gfCNCPoint4[13273] = {X 270.8909, Y 44.1700, Z -5.5000, A 0.000, B 0.000, C 0.000 }
gfCNCPoint4[13274] = {X 270.8910, Y 45.0000, Z -5.5000, A 0.000, B 0.000, C 0.000 }
gfCNCPoint4[13275] = {X 270.7867, Y 45.9257, Z -5.5000, A 0.000, B 0.000, C 0.000 }
gfCNCPoint4[13276] = {X 270.4791, Y 46.8050, Z -5.5000, A 0.000, B 0.000, C 0.000 }
gfCNCPoint4[13277] = {X 269.9835, Y 47.5937, Z -5.5000, A 0.000, B 0.000, C 0.000 }
gfCNCPoint4[13278] = {X 269.3247, Y 48.2524, Z -5.5000, A 0.000, B 0.000, C 0.000 }
gfCNCPoint4[13279] = {X 268.5360, Y 48.7480, Z -5.5000, A 0.000, B 0.000, C 0.000 }
gfCNCPoint4[13280] = {X 267.6567, Y 49.0557, Z -5.5000, A 0.000, B 0.000, C 0.000 }
gfCNCPoint4[13281] = {X 266.7310, Y 49.1600, Z -5.5000, A 0.000, B 0.000, C 0.000 }
gfCNCPoint4[13282] = {X 260.2876, Y 49.1600, Z -5.5000, A 0.000, B 0.000, C 0.000 }
gfCNCPoint4[13283] = {X 259.3664, Y 49.0567, Z -5.5000, A 0.000, B 0.000, C 0.000 }
gfCNCPoint4[13284] = {X 258.4910, Y 48.7520, Z -5.5000, A 0.000, B 0.000, C 0.000 }
gfCNCPoint4[13285] = {X 257.7047, Y 48.2611, Z -5.5000, A 0.000, B 0.000, C 0.000 }
gfCNCPoint4[13286] = {X 257.0467, Y 47.6082, Z -5.5000, A 0.000, B 0.000, C 0.000 }
gfCNCPoint4[13287] = {X 256.5496, Y 46.8258, Z -5.5000, A 0.000, B 0.000, C 0.000 }
gfCNCPoint4[13288] = {X 256.2381, Y 45.9527, Z -5.5000, A 0.000, B 0.000, C 0.000 }
gfCNCPoint4[13289] = {X 256.1277, Y 45.0324, Z -5.5000, A 0.000, B 0.000, C 0.000 }
gfCNCPoint4[13290] = {X 256.1280, Y 44.1516, Z -5.5000, A 0.000, B 0.000, C 0.000 }
gfCNCPoint4[13291] = {X 256.2385, Y 43.2545, Z -5.5000, A 0.000, B 0.000, C 0.000 }
gfCNCPoint4[13292] = {X 256.5401, Y 42.4026, Z -5.5000, A 0.000, B 0.000, C 0.000 }
gfCNCPoint4[13293] = {X 257.0187, Y 41.6358, Z -5.5000, A 0.000, B 0.000, C 0.000 }
gfCNCPoint4[13294] = {X 257.6515, Y 40.9906, Z -5.5000, A 0.000, B 0.000, C 0.000 }
gfCNCPoint4[13295] = {X 257.6515, Y 34.3138, Z -5.5000, A 0.000, B 0.000, C 0.000 }
gfCNCPoint4[13296] = {X 254.6703, Y 34.3138, Z -5.5000, A 0.000, B 0.000, C 0.000 }
gfCNCPoint4[13297] = {X 250.3102, Y 42.8068, Z -5.5000, A 0.000, B 0.000, C 0.000 }
gfCNCPoint4[13298] = {X 250.4892, Y 43.4800, Z -5.5000, A 0.000, B 0.000, C 0.000 }
gfCNCPoint4[13299] = {X 250.5534, Y 44.1736, Z -5.5000, A 0.000, B 0.000, C 0.000 }
gfCNCPoint4[13300] = {X 250.5536, Y 45.0000, Z -5.5000, A 0.000, B 0.000, C 0.000 }
gfCNCPoint4[13301] = {X 250.4493, Y 45.9257, Z -5.5000, A 0.000, B 0.000, C 0.000 }
gfCNCPoint4[13302] = {X 250.1416, Y 46.8050, Z -5.5000, A 0.000, B 0.000, C 0.000 }
gfCNCPoint4[13303] = {X 249.6460, Y 47.5937, Z -5.5000, A 0.000, B 0.000, C 0.000 }
gfCNCPoint4[13304] = {X 248.9873, Y 48.2524, Z -5.5000, A 0.000, B 0.000, C 0.000 }
gfCNCPoint4[13305] = {X 248.1985, Y 48.7480, Z -5.5000, A 0.000, B 0.000, C 0.000 }
gfCNCPoint4[13306] = {X 247.3192, Y 49.0557, Z -5.5000, A 0.000, B 0.000, C 0.000 }
gfCNCPoint4[13307] = {X 246.3936, Y 49.1600, Z -5.5000, A 0.000, B 0.000, C 0.000 }
gfCNCPoint4[13308] = {X 239.8075, Y 49.1600, Z -5.5000, A 0.000, B 0.000, C 0.000 }
gfCNCPoint4[13309] = {X 238.8818, Y 49.0557, Z -5.5000, A 0.000, B 0.000, C 0.000 }
gfCNCPoint4[13310] = {X 238.0026, Y 48.7480, Z -5.5000, A 0.000, B 0.000, C 0.000 }
gfCNCPoint4[13311] = {X 237.2138, Y 48.2524, Z -5.5000, A 0.000, B 0.000, C 0.000 }
gfCNCPoint4[13312] = {X 236.5551, Y 47.5937, Z -5.5000, A 0.000, B 0.000, C 0.000 }
gfCNCPoint4[13313] = {X 236.0595, Y 46.8050, Z -5.5000, A 0.000, B 0.000, C 0.000 }
gfCNCPoint4[13314] = {X 235.7518, Y 45.9257, Z -5.5000, A 0.000, B 0.000, C 0.000 }
gfCNCPoint4[13315] = {X 235.6475, Y 45.0000, Z -5.5000, A 0.000, B 0.000, C 0.000 }
gfCNCPoint4[13316] = {X 235.6479, Y 44.1516, Z -5.5000, A 0.000, B 0.000, C 0.000 }
gfCNCPoint4[13317] = {X 235.7441, Y 43.3174, Z -5.5000, A 0.000, B 0.000, C 0.000 }
gfCNCPoint4[13318] = {X 236.0059, Y 42.5195, Z -5.5000, A 0.000, B 0.000, C 0.000 }
gfCNCPoint4[13319] = {X 236.4226, Y 41.7905, Z -5.5000, A 0.000, B 0.000, C 0.000 }
gfCNCPoint4[13320] = {X 236.9772, Y 41.1600, Z -5.5000, A 0.000, B 0.000, C 0.000 }
gfCNCPoint4[13321] = {X 237.6471, Y 40.6537, Z -5.5000, A 0.000, B 0.000, C 0.000 }
gfCNCPoint4[13322] = {X 238.4051, Y 40.2923, Z -5.5000, A 0.000, B 0.000, C 0.000 }
gfCNCPoint4[13323] = {X 242.4918, Y 32.2930, Z -5.5000, A 0.000, B 0.000, C 0.000 }
gfCNCPoint4[13324] = {X 241.3078, Y 31.5182, Z -5.5000, A 0.000, B 0.000, C 0.000 }
gfCNCPoint4[13325] = {X 240.2313, Y 30.5999, Z -5.5000, A 0.000, B 0.000, C 0.000 }
gfCNCPoint4[13326] = {X 239.2796, Y 29.5527, Z -5.5000, A 0.000, B 0.000, C 0.000 }
gfCNCPoint4[13327] = {X 238.4681, Y 28.3935, Z -5.5000, A 0.000, B 0.000, C 0.000 }
gfCNCPoint4[13328] = {X 237.8099, Y 27.1410, Z -5.5000, A 0.000, B 0.000, C 0.000 }
gfCNCPoint4[13329] = {X 237.3154, Y 25.8152, Z -5.5000, A 0.000, B 0.000, C 0.000 }
gfCNCPoint4[13330] = {X 236.8995, Y 24.0215, Z -5.5000, A 0.000, B 0.000, C 0.000 }
gfCNCPoint4[13331] = {X 236.6876, Y 22.1924, Z -5.5000, A 0.000, B 0.000, C 0.000 }
gfCNCPoint4[13332] = {X 236.6824, Y 20.3512, Z -5.5000, A 0.000, B 0.000, C 0.000 }
gfCNCPoint4[13333] = {X 236.8839, Y 18.5210, Z -5.5000, A 0.000, B 0.000, C 0.000 }
gfCNCPoint4[13334] = {X 237.2897, Y 16.7249, Z -5.5000, A 0.000, B 0.000, C 0.000 }
gfCNCPoint4[13335] = {X 237.8524, Y 15.1703, Z -5.5000, A 0.000, B 0.000, C 0.000 }
gfCNCPoint4[13336] = {X 238.6289, Y 13.7107, Z -5.5000, A 0.000, B 0.000, C 0.000 }
gfCNCPoint4[13337] = {X 239.6035, Y 12.3752, Z -5.5000, A 0.000, B 0.000, C 0.000 }
gfCNCPoint4[13338] = {X 240.7569, Y 11.1905, Z -5.5000, A 0.000, B 0.000, C 0.000 }
gfCNCPoint4[13339] = {X 242.0658, Y 10.1805, Z -5.5000, A 0.000, B 0.000, C 0.000 }
gfCNCPoint4[13340] = {X 243.5041, Y 9.3652, Z -5.5000, A 0.000, B 0.000, C 0.000 }
gfCNCPoint4[13341] = {X 245.0431, Y 8.7610, Z -5.5000, A 0.000, B 0.000, C 0.000 }
gfCNCPoint4[13342] = {X 246.6520, Y 8.3800, Z -5.5000, A 0.000, B 0.000, C 0.000 }
gfCNCPoint4[13343] = {X 248.7352, Y 8.1102, Z -5.5000, A 0.000, B 0.000, C 0.000 }
gfCNCPoint4[13344] = {X 250.8343, Y 8.0302, Z -5.5000, A 0.000, B 0.000, C 0.000 }
gfCNCPoint4[13345] = {X 266.7621, Y 8.0302, Z -5.5000, A 0.000, B 0.000, C 0.000 }
gfCNCPoint4[13346] = {X 267.6819, Y 8.1408, Z -5.5000, A 0.000, B 0.000, C 0.000 }
gfCNCPoint4[13347] = {X 268.5546, Y 8.4520, Z -5.5000, A 0.000, B 0.000, C 0.000 }
gfCNCPoint4[13348] = {X 269.3368, Y 8.9486, Z -5.5000, A 0.000, B 0.000, C 0.000 }
gfCNCPoint4[13349] = {X 269.9897, Y 9.6059, Z -5.5000, A 0.000, B 0.000, C 0.000 }
gfCNCPoint4[13350] = {X 270.4811, Y 10.3913, Z -5.5000, A 0.000, B 0.000, C 0.000 }
gfCNCPoint4[13351] = {X 270.7866, Y 11.2660, Z -5.5000, A 0.000, B 0.000, C 0.000 }
gfCNCPoint4[13352] = {X 270.8910, Y 12.1866, Z -5.5000, A 0.000, B 0.000, C 0.000 }
gfCNCPoint4[13353] = {X 270.8908, Y 13.0208, Z -5.5000, A 0.000, B 0.000, C 0.000 }
gfCNCPoint4[13354] = {X 270.7824, Y 13.9226, Z -5.5000, A 0.000, B 0.000, C 0.000 }
gfCNCPoint4[13355] = {X 270.4808, Y 14.7793, Z -5.5000, A 0.000, B 0.000, C 0.000 }
gfCNCPoint4[13356] = {X 270.0005, Y 15.5502, Z -5.5000, A 0.000, B 0.000, C 0.000 }
gfCNCPoint4[13357] = {X 269.3643, Y 16.1985, Z -5.5000, A 0.000, B 0.000, C 0.000 }
gfCNCPoint4[13358] = {X 269.3642, Y 28.5936, Z -5.5000, A 0.000, B 0.000, C 0.000 }
gfCNCPoint4[13359] = {X 273.3642, Y 28.5936, Z -5.5000, A 0.000, B 0.000, C 0.000 }
gfCNCPoint4[13360] = {X 269.2842, Y 28.5936, Z -5.5000, A 0.000, B 0.000, C 0.000 }
gfCNCPoint4[13361] = {X 269.2842, Y 41.0277, Z -5.5000, A 0.000, B 0.000, C 0.000 }
gfCNCPoint4[13362] = {X 269.3838, Y 41.1089, Z -5.5000, A 0.000, B 0.000, C 0.000 }
gfCNCPoint4[13363] = {X 269.9802, Y 41.7411, Z -5.5000, A 0.000, B 0.000, C 0.000 }
gfCNCPoint4[13364] = {X 270.4291, Y 42.4852, Z -5.5000, A 0.000, B 0.000, C 0.000 }
gfCNCPoint4[13365] = {X 270.7103, Y 43.3076, Z -5.5000, A 0.000, B 0.000, C 0.000 }
gfCNCPoint4[13366] = {X 270.8109, Y 44.1708, Z -5.5000, A 0.000, B 0.000, C 0.000 }
gfCNCPoint4[13367] = {X 270.8110, Y 45.0000, Z -5.5000, A 0.000, B 0.000, C 0.000 }
gfCNCPoint4[13368] = {X 270.7087, Y 45.9079, Z -5.5000, A 0.000, B 0.000, C 0.000 }
gfCNCPoint4[13369] = {X 270.4070, Y 46.7702, Z -5.5000, A 0.000, B 0.000, C 0.000 }
gfCNCPoint4[13370] = {X 269.9209, Y 47.5438, Z -5.5000, A 0.000, B 0.000, C 0.000 }
gfCNCPoint4[13371] = {X 269.2749, Y 48.1899, Z -5.5000, A 0.000, B 0.000, C 0.000 }
gfCNCPoint4[13372] = {X 268.5013, Y 48.6760, Z -5.5000, A 0.000, B 0.000, C 0.000 }
gfCNCPoint4[13373] = {X 267.6389, Y 48.9777, Z -5.5000, A 0.000, B 0.000, C 0.000 }
gfCNCPoint4[13374] = {X 266.7310, Y 49.0800, Z -5.5000, A 0.000, B 0.000, C 0.000 }
gfCNCPoint4[13375] = {X 260.2876, Y 49.0800, Z -5.5000, A 0.000, B 0.000, C 0.000 }
gfCNCPoint4[13376] = {X 259.3841, Y 48.9787, Z -5.5000, A 0.000, B 0.000, C 0.000 }
gfCNCPoint4[13377] = {X 258.5255, Y 48.6799, Z -5.5000, A 0.000, B 0.000, C 0.000 }
gfCNCPoint4[13378] = {X 257.7544, Y 48.1983, Z -5.5000, A 0.000, B 0.000, C 0.000 }
gfCNCPoint4[13379] = {X 257.1090, Y 47.5580, Z -5.5000, A 0.000, B 0.000, C 0.000 }
gfCNCPoint4[13380] = {X 256.6215, Y 46.7907, Z -5.5000, A 0.000, B 0.000, C 0.000 }
gfCNCPoint4[13381] = {X 256.3160, Y 45.9344, Z -5.5000, A 0.000, B 0.000, C 0.000 }
gfCNCPoint4[13382] = {X 256.2077, Y 45.0318, Z -5.5000, A 0.000, B 0.000, C 0.000 }
gfCNCPoint4[13383] = {X 256.2080, Y 44.1527, Z -5.5000, A 0.000, B 0.000, C 0.000 }
gfCNCPoint4[13384] = {X 256.3185, Y 43.2637, Z -5.5000, A 0.000, B 0.000, C 0.000 }
gfCNCPoint4[13385] = {X 256.6204, Y 42.4203, Z -5.5000, A 0.000, B 0.000, C 0.000 }
gfCNCPoint4[13386] = {X 257.0991, Y 41.6631, Z -5.5000, A 0.000, B 0.000, C 0.000 }
gfCNCPoint4[13387] = {X 257.7315, Y 41.0287, Z -5.5000, A 0.000, B 0.000, C 0.000 }
gfCNCPoint4[13388] = {X 257.7315, Y 34.2338, Z -5.5000, A 0.000, B 0.000, C 0.000 }
gfCNCPoint4[13389] = {X 254.6215, Y 34.2338, Z -5.5000, A 0.000, B 0.000, C 0.000 }
gfCNCPoint4[13390] = {X 250.2231, Y 42.8013, Z -5.5000, A 0.000, B 0.000, C 0.000 }
gfCNCPoint4[13391] = {X 250.4074, Y 43.4770, Z -5.5000, A 0.000, B 0.000, C 0.000 }
gfCNCPoint4[13392] = {X 250.4734, Y 44.1743, Z -5.5000, A 0.000, B 0.000, C 0.000 }
gfCNCPoint4[13393] = {X 250.4736, Y 45.0000, Z -5.5000, A 0.000, B 0.000, C 0.000 }
gfCNCPoint4[13394] = {X 250.3713, Y 45.9079, Z -5.5000, A 0.000, B 0.000, C 0.000 }
gfCNCPoint4[13395] = {X 250.0695, Y 46.7702, Z -5.5000, A 0.000, B 0.000, C 0.000 }
gfCNCPoint4[13396] = {X 249.5834, Y 47.5438, Z -5.5000, A 0.000, B 0.000, C 0.000 }
gfCNCPoint4[13397] = {X 248.9374, Y 48.1899, Z -5.5000, A 0.000, B 0.000, C 0.000 }
gfCNCPoint4[13398] = {X 248.1638, Y 48.6760, Z -5.5000, A 0.000, B 0.000, C 0.000 }
gfCNCPoint4[13399] = {X 247.3014, Y 48.9777, Z -5.5000, A 0.000, B 0.000, C 0.000 }
gfCNCPoint4[13400] = {X 246.3936, Y 49.0800, Z -5.5000, A 0.000, B 0.000, C 0.000 }
gfCNCPoint4[13401] = {X 239.8075, Y 49.0800, Z -5.5000, A 0.000, B 0.000, C 0.000 }
gfCNCPoint4[13402] = {X 238.8996, Y 48.9777, Z -5.5000, A 0.000, B 0.000, C 0.000 }
gfCNCPoint4[13403] = {X 238.0373, Y 48.6760, Z -5.5000, A 0.000, B 0.000, C 0.000 }
gfCNCPoint4[13404] = {X 237.2637, Y 48.1899, Z -5.5000, A 0.000, B 0.000, C 0.000 }
gfCNCPoint4[13405] = {X 236.6176, Y 47.5438, Z -5.5000, A 0.000, B 0.000, C 0.000 }
gfCNCPoint4[13406] = {X 236.1315, Y 46.7702, Z -5.5000, A 0.000, B 0.000, C 0.000 }
gfCNCPoint4[13407] = {X 235.8298, Y 45.9079, Z -5.5000, A 0.000, B 0.000, C 0.000 }
gfCNCPoint4[13408] = {X 235.7275, Y 45.0000, Z -5.5000, A 0.000, B 0.000, C 0.000 }
gfCNCPoint4[13409] = {X 235.7279, Y 44.1527, Z -5.5000, A 0.000, B 0.000, C 0.000 }
gfCNCPoint4[13410] = {X 235.8234, Y 43.3294, Z -5.5000, A 0.000, B 0.000, C 0.000 }
gfCNCPoint4[13411] = {X 236.0833, Y 42.5424, Z -5.5000, A 0.000, B 0.000, C 0.000 }
gfCNCPoint4[13412] = {X 236.4969, Y 41.8242, Z -5.5000, A 0.000, B 0.000, C 0.000 }
gfCNCPoint4[13413] = {X 237.0471, Y 41.2044, Z -5.5000, A 0.000, B 0.000, C 0.000 }
gfCNCPoint4[13414] = {X 237.7112, Y 40.7085, Z -5.5000, A 0.000, B 0.000, C 0.000 }
gfCNCPoint4[13415] = {X 238.4618, Y 40.3571, Z -5.5000, A 0.000, B 0.000, C 0.000 }
gfCNCPoint4[13416] = {X 242.5980, Y 32.2609, Z -5.5000, A 0.000, B 0.000, C 0.000 }
gfCNCPoint4[13417] = {X 241.4069, Y 31.4923, Z -5.5000, A 0.000, B 0.000, C 0.000 }
gfCNCPoint4[13418] = {X 240.3237, Y 30.5779, Z -5.5000, A 0.000, B 0.000, C 0.000 }
gfCNCPoint4[13419] = {X 239.3661, Y 29.5326, Z -5.5000, A 0.000, B 0.000, C 0.000 }
gfCNCPoint4[13420] = {X 238.5498, Y 28.3737, Z -5.5000, A 0.000, B 0.000, C 0.000 }
gfCNCPoint4[13421] = {X 237.8881, Y 27.1200, Z -5.5000, A 0.000, B 0.000, C 0.000 }
gfCNCPoint4[13422] = {X 237.3920, Y 25.7920, Z -5.5000, A 0.000, B 0.000, C 0.000 }
gfCNCPoint4[13423] = {X 236.9782, Y 24.0072, Z -5.5000, A 0.000, B 0.000, C 0.000 }
gfCNCPoint4[13424] = {X 236.7675, Y 22.1872, Z -5.5000, A 0.000, B 0.000, C 0.000 }
gfCNCPoint4[13425] = {X 236.7623, Y 20.3551, Z -5.5000, A 0.000, B 0.000, C 0.000 }
gfCNCPoint4[13426] = {X 236.9629, Y 18.5340, Z -5.5000, A 0.000, B 0.000, C 0.000 }
gfCNCPoint4[13427] = {X 237.3666, Y 16.7469, Z -5.5000, A 0.000, B 0.000, C 0.000 }
gfCNCPoint4[13428] = {X 237.9255, Y 15.2028, Z -5.5000, A 0.000, B 0.000, C 0.000 }
gfCNCPoint4[13429] = {X 238.6967, Y 13.7531, Z -5.5000, A 0.000, B 0.000, C 0.000 }
gfCNCPoint4[13430] = {X 239.6648, Y 12.4267, Z -5.5000, A 0.000, B 0.000, C 0.000 }
gfCNCPoint4[13431] = {X 240.8103, Y 11.2501, Z -5.5000, A 0.000, B 0.000, C 0.000 }
gfCNCPoint4[13432] = {X 242.1103, Y 10.2469, Z -5.5000, A 0.000, B 0.000, C 0.000 }
gfCNCPoint4[13433] = {X 243.5389, Y 9.4372, Z -5.5000, A 0.000, B 0.000, C 0.000 }
gfCNCPoint4[13434] = {X 245.0674, Y 8.8372, Z -5.5000, A 0.000, B 0.000, C 0.000 }
gfCNCPoint4[13435] = {X 246.6654, Y 8.4589, Z -5.5000, A 0.000, B 0.000, C 0.000 }
gfCNCPoint4[13436] = {X 248.7418, Y 8.1900, Z -5.5000, A 0.000, B 0.000, C 0.000 }
gfCNCPoint4[13437] = {X 250.8340, Y 8.1102, Z -5.5000, A 0.000, B 0.000, C 0.000 }
gfCNCPoint4[13438] = {X 266.7614, Y 8.1102, Z -5.5000, A 0.000, B 0.000, C 0.000 }
gfCNCPoint4[13439] = {X 267.6636, Y 8.2186, Z -5.5000, A 0.000, B 0.000, C 0.000 }
gfCNCPoint4[13440] = {X 268.5195, Y 8.5239, Z -5.5000, A 0.000, B 0.000, C 0.000 }
gfCNCPoint4[13441] = {X 269.2866, Y 9.0109, Z -5.5000, A 0.000, B 0.000, C 0.000 }
gfCNCPoint4[13442] = {X 269.9271, Y 9.6556, Z -5.5000, A 0.000, B 0.000, C 0.000 }
gfCNCPoint4[13443] = {X 270.4090, Y 10.4260, Z -5.5000, A 0.000, B 0.000, C 0.000 }
gfCNCPoint4[13444] = {X 270.7086, Y 11.2838, Z -5.5000, A 0.000, B 0.000, C 0.000 }
gfCNCPoint4[13445] = {X 270.8110, Y 12.1867, Z -5.5000, A 0.000, B 0.000, C 0.000 }
gfCNCPoint4[13446] = {X 270.8108, Y 13.0200, Z -5.5000, A 0.000, B 0.000, C 0.000 }
gfCNCPoint4[13447] = {X 270.7023, Y 13.9136, Z -5.5000, A 0.000, B 0.000, C 0.000 }
gfCNCPoint4[13448] = {X 270.4005, Y 14.7617, Z -5.5000, A 0.000, B 0.000, C 0.000 }
gfCNCPoint4[13449] = {X 269.9200, Y 15.5230, Z -5.5000, A 0.000, B 0.000, C 0.000 }
gfCNCPoint4[13450] = {X 269.2843, Y 16.1603, Z -5.5000, A 0.000, B 0.000, C 0.000 }
gfCNCPoint4[13451] = {X 269.2842, Y 28.5936, Z -5.5000, A 0.000, B 0.000, C 0.000 }
gfCNCPoint4[13452] = {X 273.2842, Y 28.5936, Z -5.5000, A 0.000, B 0.000, C 0.000 }
gfCNCPoint4[13453] = {X 269.2042, Y 28.5936, Z -5.5000, A 0.000, B 0.000, C 0.000 }
gfCNCPoint4[13454] = {X 269.2042, Y 41.0656, Z -5.5000, A 0.000, B 0.000, C 0.000 }
gfCNCPoint4[13455] = {X 269.3430, Y 41.1793, Z -5.5000, A 0.000, B 0.000, C 0.000 }
gfCNCPoint4[13456] = {X 269.9287, Y 41.8057, Z -5.5000, A 0.000, B 0.000, C 0.000 }
gfCNCPoint4[13457] = {X 270.3675, Y 42.5427, Z -5.5000, A 0.000, B 0.000, C 0.000 }
gfCNCPoint4[13458] = {X 270.6391, Y 43.3562, Z -5.5000, A 0.000, B 0.000, C 0.000 }
gfCNCPoint4[13459] = {X 270.7310, Y 44.2089, Z -5.5000, A 0.000, B 0.000, C 0.000 }
gfCNCPoint4[13460] = {X 270.7310, Y 45.0000, Z -5.5000, A 0.000, B 0.000, C 0.000 }
gfCNCPoint4[13461] = {X 270.6307, Y 45.8901, Z -5.5000, A 0.000, B 0.000, C 0.000 }
gfCNCPoint4[13462] = {X 270.3349, Y 46.7355, Z -5.5000, A 0.000, B 0.000, C 0.000 }
gfCNCPoint4[13463] = {X 269.8584, Y 47.4940, Z -5.5000, A 0.000, B 0.000, C 0.000 }
gfCNCPoint4[13464] = {X 269.2250, Y 48.1273, Z -5.5000, A 0.000, B 0.000, C 0.000 }
gfCNCPoint4[13465] = {X 268.4666, Y 48.6039, Z -5.5000, A 0.000, B 0.000, C 0.000 }
gfCNCPoint4[13466] = {X 267.6211, Y 48.8997, Z -5.5000, A 0.000, B 0.000, C 0.000 }
gfCNCPoint4[13467] = {X 266.7310, Y 49.0000, Z -5.5000, A 0.000, B 0.000, C 0.000 }
gfCNCPoint4[13468] = {X 260.2876, Y 49.0000, Z -5.5000, A 0.000, B 0.000, C 0.000 }
gfCNCPoint4[13469] = {X 259.3975, Y 48.8997, Z -5.5000, A 0.000, B 0.000, C 0.000 }
gfCNCPoint4[13470] = {X 258.5520, Y 48.6039, Z -5.5000, A 0.000, B 0.000, C 0.000 }
gfCNCPoint4[13471] = {X 257.7936, Y 48.1273, Z -5.5000, A 0.000, B 0.000, C 0.000 }
gfCNCPoint4[13472] = {X 257.1602, Y 47.4939, Z -5.5000, A 0.000, B 0.000, C 0.000 }
gfCNCPoint4[13473] = {X 256.6837, Y 46.7355, Z -5.5000, A 0.000, B 0.000, C 0.000 }
gfCNCPoint4[13474] = {X 256.3878, Y 45.8901, Z -5.5000, A 0.000, B 0.000, C 0.000 }
gfCNCPoint4[13475] = {X 256.2876, Y 45.0000, Z -5.5000, A 0.000, B 0.000, C 0.000 }
gfCNCPoint4[13476] = {X 256.2879, Y 44.1538, Z -5.5000, A 0.000, B 0.000, C 0.000 }
gfCNCPoint4[13477] = {X 256.3986, Y 43.2730, Z -5.5000, A 0.000, B 0.000, C 0.000 }
gfCNCPoint4[13478] = {X 256.7008, Y 42.4382, Z -5.5000, A 0.000, B 0.000, C 0.000 }
gfCNCPoint4[13479] = {X 257.1796, Y 41.6907, Z -5.5000, A 0.000, B 0.000, C 0.000 }
gfCNCPoint4[13480] = {X 257.8115, Y 41.0672, Z -5.5000, A 0.000, B 0.000, C 0.000 }
gfCNCPoint4[13481] = {X 257.8115, Y 34.1538, Z -5.5000, A 0.000, B 0.000, C 0.000 }
gfCNCPoint4[13482] = {X 254.8169, Y 34.1538, Z -5.5000, A 0.000, B 0.000, C 0.000 }
gfCNCPoint4[13483] = {X 254.5733, Y 34.1525, Z -5.5000, A 0.000, B 0.000, C 0.000 }
gfCNCPoint4[13484] = {X 250.1358, Y 42.7961, Z -5.5000, A 0.000, B 0.000, C 0.000 }
gfCNCPoint4[13485] = {X 250.3286, Y 43.4908, Z -5.5000, A 0.000, B 0.000, C 0.000 }
gfCNCPoint4[13486] = {X 250.3936, Y 44.2089, Z -5.5000, A 0.000, B 0.000, C 0.000 }
gfCNCPoint4[13487] = {X 250.3936, Y 45.0000, Z -5.5000, A 0.000, B 0.000, C 0.000 }
gfCNCPoint4[13488] = {X 250.2933, Y 45.8901, Z -5.5000, A 0.000, B 0.000, C 0.000 }
gfCNCPoint4[13489] = {X 249.9974, Y 46.7355, Z -5.5000, A 0.000, B 0.000, C 0.000 }
gfCNCPoint4[13490] = {X 249.5209, Y 47.4940, Z -5.5000, A 0.000, B 0.000, C 0.000 }
gfCNCPoint4[13491] = {X 248.8875, Y 48.1273, Z -5.5000, A 0.000, B 0.000, C 0.000 }
gfCNCPoint4[13492] = {X 248.1291, Y 48.6039, Z -5.5000, A 0.000, B 0.000, C 0.000 }
gfCNCPoint4[13493] = {X 247.2836, Y 48.8997, Z -5.5000, A 0.000, B 0.000, C 0.000 }
gfCNCPoint4[13494] = {X 246.3936, Y 49.0000, Z -5.5000, A 0.000, B 0.000, C 0.000 }
gfCNCPoint4[13495] = {X 239.8075, Y 49.0000, Z -5.5000, A 0.000, B 0.000, C 0.000 }
gfCNCPoint4[13496] = {X 238.9174, Y 48.8997, Z -5.5000, A 0.000, B 0.000, C 0.000 }
gfCNCPoint4[13497] = {X 238.0720, Y 48.6039, Z -5.5000, A 0.000, B 0.000, C 0.000 }
gfCNCPoint4[13498] = {X 237.3135, Y 48.1273, Z -5.5000, A 0.000, B 0.000, C 0.000 }
gfCNCPoint4[13499] = {X 236.6802, Y 47.4940, Z -5.5000, A 0.000, B 0.000, C 0.000 }
gfCNCPoint4[13500] = {X 236.2036, Y 46.7355, Z -5.5000, A 0.000, B 0.000, C 0.000 }
gfCNCPoint4[13501] = {X 235.9078, Y 45.8901, Z -5.5000, A 0.000, B 0.000, C 0.000 }
gfCNCPoint4[13502] = {X 235.8075, Y 45.0000, Z -5.5000, A 0.000, B 0.000, C 0.000 }
gfCNCPoint4[13503] = {X 235.8079, Y 44.1538, Z -5.5000, A 0.000, B 0.000, C 0.000 }
gfCNCPoint4[13504] = {X 235.9027, Y 43.3414, Z -5.5000, A 0.000, B 0.000, C 0.000 }
gfCNCPoint4[13505] = {X 236.1607, Y 42.5654, Z -5.5000, A 0.000, B 0.000, C 0.000 }
gfCNCPoint4[13506] = {X 236.5712, Y 41.8580, Z -5.5000, A 0.000, B 0.000, C 0.000 }
gfCNCPoint4[13507] = {X 237.1169, Y 41.2489, Z -5.5000, A 0.000, B 0.000, C 0.000 }
gfCNCPoint4[13508] = {X 237.7752, Y 40.7635, Z -5.5000, A 0.000, B 0.000, C 0.000 }
gfCNCPoint4[13509] = {X 238.5184, Y 40.4222, Z -5.5000, A 0.000, B 0.000, C 0.000 }
gfCNCPoint4[13510] = {X 242.7045, Y 32.2284, Z -5.5000, A 0.000, B 0.000, C 0.000 }
gfCNCPoint4[13511] = {X 241.5063, Y 31.4661, Z -5.5000, A 0.000, B 0.000, C 0.000 }
gfCNCPoint4[13512] = {X 240.4162, Y 30.5557, Z -5.5000, A 0.000, B 0.000, C 0.000 }
gfCNCPoint4[13513] = {X 239.4526, Y 29.5125, Z -5.5000, A 0.000, B 0.000, C 0.000 }
gfCNCPoint4[13514] = {X 238.6314, Y 28.3538, Z -5.5000, A 0.000, B 0.000, C 0.000 }
gfCNCPoint4[13515] = {X 237.9664, Y 27.0989, Z -5.5000, A 0.000, B 0.000, C 0.000 }
gfCNCPoint4[13516] = {X 237.4686, Y 25.7689, Z -5.5000, A 0.000, B 0.000, C 0.000 }
gfCNCPoint4[13517] = {X 237.0570, Y 23.9929, Z -5.5000, A 0.000, B 0.000, C 0.000 }
gfCNCPoint4[13518] = {X 236.8473, Y 22.1820, Z -5.5000, A 0.000, B 0.000, C 0.000 }
gfCNCPoint4[13519] = {X 236.8422, Y 20.3590, Z -5.5000, A 0.000, B 0.000, C 0.000 }
gfCNCPoint4[13520] = {X 237.0418, Y 18.5469, Z -5.5000, A 0.000, B 0.000, C 0.000 }
gfCNCPoint4[13521] = {X 237.4436, Y 16.7687, Z -5.5000, A 0.000, B 0.000, C 0.000 }
gfCNCPoint4[13522] = {X 237.9987, Y 15.2353, Z -5.5000, A 0.000, B 0.000, C 0.000 }
gfCNCPoint4[13523] = {X 238.7646, Y 13.7955, Z -5.5000, A 0.000, B 0.000, C 0.000 }
gfCNCPoint4[13524] = {X 239.7260, Y 12.4782, Z -5.5000, A 0.000, B 0.000, C 0.000 }
gfCNCPoint4[13525] = {X 240.8637, Y 11.3097, Z -5.5000, A 0.000, B 0.000, C 0.000 }
gfCNCPoint4[13526] = {X 242.1548, Y 10.3134, Z -5.5000, A 0.000, B 0.000, C 0.000 }
gfCNCPoint4[13527] = {X 243.5737, Y 9.5093, Z -5.5000, A 0.000, B 0.000, C 0.000 }
gfCNCPoint4[13528] = {X 245.0918, Y 8.9134, Z -5.5000, A 0.000, B 0.000, C 0.000 }
gfCNCPoint4[13529] = {X 246.6787, Y 8.5377, Z -5.5000, A 0.000, B 0.000, C 0.000 }
gfCNCPoint4[13530] = {X 248.7483, Y 8.2697, Z -5.5000, A 0.000, B 0.000, C 0.000 }
gfCNCPoint4[13531] = {X 250.8336, Y 8.1902, Z -5.5000, A 0.000, B 0.000, C 0.000 }
gfCNCPoint4[13532] = {X 266.7608, Y 8.1902, Z -5.5000, A 0.000, B 0.000, C 0.000 }
gfCNCPoint4[13533] = {X 267.6453, Y 8.2965, Z -5.5000, A 0.000, B 0.000, C 0.000 }
gfCNCPoint4[13534] = {X 268.4844, Y 8.5958, Z -5.5000, A 0.000, B 0.000, C 0.000 }
gfCNCPoint4[13535] = {X 269.2365, Y 9.0733, Z -5.5000, A 0.000, B 0.000, C 0.000 }
gfCNCPoint4[13536] = {X 269.8644, Y 9.7053, Z -5.5000, A 0.000, B 0.000, C 0.000 }
gfCNCPoint4[13537] = {X 270.3369, Y 10.4606, Z -5.5000, A 0.000, B 0.000, C 0.000 }
gfCNCPoint4[13538] = {X 270.6306, Y 11.3017, Z -5.5000, A 0.000, B 0.000, C 0.000 }
gfCNCPoint4[13539] = {X 270.7310, Y 12.1869, Z -5.5000, A 0.000, B 0.000, C 0.000 }
gfCNCPoint4[13540] = {X 270.7308, Y 13.0192, Z -5.5000, A 0.000, B 0.000, C 0.000 }
gfCNCPoint4[13541] = {X 270.6222, Y 13.9046, Z -5.5000, A 0.000, B 0.000, C 0.000 }
gfCNCPoint4[13542] = {X 270.3201, Y 14.7439, Z -5.5000, A 0.000, B 0.000, C 0.000 }
gfCNCPoint4[13543] = {X 269.8395, Y 15.4954, Z -5.5000, A 0.000, B 0.000, C 0.000 }
gfCNCPoint4[13544] = {X 269.2043, Y 16.1217, Z -5.5000, A 0.000, B 0.000, C 0.000 }
gfCNCPoint4[13545] = {X 269.2042, Y 28.5936, Z -5.5000, A 0.000, B 0.000, C 0.000 }
gfCNCPoint4[13546] = {X 273.2842, Y 28.5936, Z -5.5000, A 0.000, B 0.000, C 0.000 }
gfCNCPoint4[13547] = {X 273.2842, Y 28.5936, Z -2.5000, A 0.000, B 0.000, C 0.000 }
gfCNCPoint4[13548] = {X 273.2842, Y 28.5936, Z 11.0000, A 0.000, B 0.000, C 0.000 }
gfCNCPoint4[13549] = {X 277.7448, Y 28.5923, Z 11.0000, A 0.000, B 0.000, C 0.000 }
gfCNCPoint4[13550] = {X 277.7448, Y 28.5923, Z -2.5000, A 0.000, B 0.000, C 0.000 }
gfCNCPoint4[13551] = {X 277.7448, Y 28.5923, Z -5.5000, A 0.000, B 0.000, C 0.000 }
gfCNCPoint4[13552] = {X 281.8248, Y 28.5922, Z -5.5000, A 0.000, B 0.000, C 0.000 }
gfCNCPoint4[13553] = {X 281.8246, Y 16.2737, Z -5.5000, A 0.000, B 0.000, C 0.000 }
gfCNCPoint4[13554] = {X 281.1863, Y 15.6026, Z -5.5000, A 0.000, B 0.000, C 0.000 }
gfCNCPoint4[13555] = {X 280.7058, Y 14.8109, Z -5.5000, A 0.000, B 0.000, C 0.000 }
gfCNCPoint4[13556] = {X 280.4050, Y 13.9349, Z -5.5000, A 0.000, B 0.000, C 0.000 }
gfCNCPoint4[13557] = {X 280.2978, Y 13.0150, Z -5.5000, A 0.000, B 0.000, C 0.000 }
gfCNCPoint4[13558] = {X 280.2977, Y 12.1868, Z -5.5000, A 0.000, B 0.000, C 0.000 }
gfCNCPoint4[13559] = {X 280.4060, Y 11.2255, Z -5.5000, A 0.000, B 0.000, C 0.000 }
gfCNCPoint4[13560] = {X 280.7255, Y 10.3124, Z -5.5000, A 0.000, B 0.000, C 0.000 }
gfCNCPoint4[13561] = {X 281.2402, Y 9.4933, Z -5.5000, A 0.000, B 0.000, C 0.000 }
gfCNCPoint4[13562] = {X 281.9242, Y 8.8093, Z -5.5000, A 0.000, B 0.000, C 0.000 }
gfCNCPoint4[13563] = {X 282.7433, Y 8.2946, Z -5.5000, A 0.000, B 0.000, C 0.000 }
gfCNCPoint4[13564] = {X 283.6564, Y 7.9751, Z -5.5000, A 0.000, B 0.000, C 0.000 }
gfCNCPoint4[13565] = {X 284.6177, Y 7.8668, Z -5.5000, A 0.000, B 0.000, C 0.000 }
gfCNCPoint4[13566] = {X 291.0611, Y 7.8668, Z -5.5000, A 0.000, B 0.000, C 0.000 }
gfCNCPoint4[13567] = {X 292.0224, Y 7.9751, Z -5.5000, A 0.000, B 0.000, C 0.000 }
gfCNCPoint4[13568] = {X 292.9355, Y 8.2946, Z -5.5000, A 0.000, B 0.000, C 0.000 }
gfCNCPoint4[13569] = {X 293.7546, Y 8.8093, Z -5.5000, A 0.000, B 0.000, C 0.000 }
gfCNCPoint4[13570] = {X 294.4386, Y 9.4933, Z -5.5000, A 0.000, B 0.000, C 0.000 }
gfCNCPoint4[13571] = {X 294.9533, Y 10.3124, Z -5.5000, A 0.000, B 0.000, C 0.000 }
gfCNCPoint4[13572] = {X 295.2728, Y 11.2255, Z -5.5000, A 0.000, B 0.000, C 0.000 }
gfCNCPoint4[13573] = {X 295.3811, Y 12.1868, Z -5.5000, A 0.000, B 0.000, C 0.000 }
gfCNCPoint4[13574] = {X 295.3811, Y 12.9782, Z -5.5000, A 0.000, B 0.000, C 0.000 }
gfCNCPoint4[13575] = {X 295.2798, Y 13.9080, Z -5.5000, A 0.000, B 0.000, C 0.000 }
gfCNCPoint4[13576] = {X 294.9806, Y 14.7941, Z -5.5000, A 0.000, B 0.000, C 0.000 }
gfCNCPoint4[13577] = {X 294.4978, Y 15.5952, Z -5.5000, A 0.000, B 0.000, C 0.000 }
gfCNCPoint4[13578] = {X 293.8539, Y 16.2735, Z -5.5000, A 0.000, B 0.000, C 0.000 }
gfCNCPoint4[13579] = {X 293.8549, Y 22.1965, Z -5.5000, A 0.000, B 0.000, C 0.000 }
gfCNCPoint4[13580] = {X 302.7589, Y 22.1965, Z -5.5000, A 0.000, B 0.000, C 0.000 }
gfCNCPoint4[13581] = {X 302.7639, Y 16.2776, Z -5.5000, A 0.000, B 0.000, C 0.000 }
gfCNCPoint4[13582] = {X 302.1239, Y 15.6065, Z -5.5000, A 0.000, B 0.000, C 0.000 }
gfCNCPoint4[13583] = {X 301.6420, Y 14.8143, Z -5.5000, A 0.000, B 0.000, C 0.000 }
gfCNCPoint4[13584] = {X 301.3402, Y 13.9375, Z -5.5000, A 0.000, B 0.000, C 0.000 }
gfCNCPoint4[13585] = {X 301.2324, Y 13.0165, Z -5.5000, A 0.000, B 0.000, C 0.000 }
gfCNCPoint4[13586] = {X 301.2323, Y 12.1868, Z -5.5000, A 0.000, B 0.000, C 0.000 }
gfCNCPoint4[13587] = {X 301.3406, Y 11.2255, Z -5.5000, A 0.000, B 0.000, C 0.000 }
gfCNCPoint4[13588] = {X 301.6601, Y 10.3124, Z -5.5000, A 0.000, B 0.000, C 0.000 }
gfCNCPoint4[13589] = {X 302.1747, Y 9.4933, Z -5.5000, A 0.000, B 0.000, C 0.000 }
gfCNCPoint4[13590] = {X 302.8588, Y 8.8093, Z -5.5000, A 0.000, B 0.000, C 0.000 }
gfCNCPoint4[13591] = {X 303.6779, Y 8.2946, Z -5.5000, A 0.000, B 0.000, C 0.000 }
gfCNCPoint4[13592] = {X 304.5910, Y 7.9751, Z -5.5000, A 0.000, B 0.000, C 0.000 }
gfCNCPoint4[13593] = {X 305.5523, Y 7.8668, Z -5.5000, A 0.000, B 0.000, C 0.000 }
gfCNCPoint4[13594] = {X 311.9957, Y 7.8668, Z -5.5000, A 0.000, B 0.000, C 0.000 }
gfCNCPoint4[13595] = {X 312.9570, Y 7.9751, Z -5.5000, A 0.000, B 0.000, C 0.000 }
gfCNCPoint4[13596] = {X 313.8701, Y 8.2946, Z -5.5000, A 0.000, B 0.000, C 0.000 }
gfCNCPoint4[13597] = {X 314.6892, Y 8.8093, Z -5.5000, A 0.000, B 0.000, C 0.000 }
gfCNCPoint4[13598] = {X 315.3732, Y 9.4933, Z -5.5000, A 0.000, B 0.000, C 0.000 }
gfCNCPoint4[13599] = {X 315.8879, Y 10.3124, Z -5.5000, A 0.000, B 0.000, C 0.000 }
gfCNCPoint4[13600] = {X 316.2074, Y 11.2255, Z -5.5000, A 0.000, B 0.000, C 0.000 }
gfCNCPoint4[13601] = {X 316.3157, Y 12.1868, Z -5.5000, A 0.000, B 0.000, C 0.000 }
gfCNCPoint4[13602] = {X 316.3157, Y 12.9782, Z -5.5000, A 0.000, B 0.000, C 0.000 }
gfCNCPoint4[13603] = {X 316.2145, Y 13.9077, Z -5.5000, A 0.000, B 0.000, C 0.000 }
gfCNCPoint4[13604] = {X 315.9156, Y 14.7937, Z -5.5000, A 0.000, B 0.000, C 0.000 }
gfCNCPoint4[13605] = {X 315.4331, Y 15.5947, Z -5.5000, A 0.000, B 0.000, C 0.000 }
gfCNCPoint4[13606] = {X 314.7895, Y 16.2730, Z -5.5000, A 0.000, B 0.000, C 0.000 }
gfCNCPoint4[13607] = {X 314.7884, Y 40.9128, Z -5.5000, A 0.000, B 0.000, C 0.000 }
gfCNCPoint4[13608] = {X 315.4268, Y 41.5838, Z -5.5000, A 0.000, B 0.000, C 0.000 }
gfCNCPoint4[13609] = {X 315.9074, Y 42.3755, Z -5.5000, A 0.000, B 0.000, C 0.000 }
gfCNCPoint4[13610] = {X 316.2083, Y 43.2514, Z -5.5000, A 0.000, B 0.000, C 0.000 }
gfCNCPoint4[13611] = {X 316.3156, Y 44.1713, Z -5.5000, A 0.000, B 0.000, C 0.000 }
gfCNCPoint4[13612] = {X 316.3157, Y 45.0000, Z -5.5000, A 0.000, B 0.000, C 0.000 }
gfCNCPoint4[13613] = {X 316.2074, Y 45.9613, Z -5.5000, A 0.000, B 0.000, C 0.000 }
gfCNCPoint4[13614] = {X 315.8879, Y 46.8744, Z -5.5000, A 0.000, B 0.000, C 0.000 }
gfCNCPoint4[13615] = {X 315.3732, Y 47.6935, Z -5.5000, A 0.000, B 0.000, C 0.000 }
gfCNCPoint4[13616] = {X 314.6892, Y 48.3775, Z -5.5000, A 0.000, B 0.000, C 0.000 }
gfCNCPoint4[13617] = {X 313.8701, Y 48.8922, Z -5.5000, A 0.000, B 0.000, C 0.000 }
gfCNCPoint4[13618] = {X 312.9570, Y 49.2117, Z -5.5000, A 0.000, B 0.000, C 0.000 }
gfCNCPoint4[13619] = {X 311.9957, Y 49.3200, Z -5.5000, A 0.000, B 0.000, C 0.000 }
gfCNCPoint4[13620] = {X 305.5523, Y 49.3200, Z -5.5000, A 0.000, B 0.000, C 0.000 }
gfCNCPoint4[13621] = {X 304.5958, Y 49.2128, Z -5.5000, A 0.000, B 0.000, C 0.000 }
gfCNCPoint4[13622] = {X 303.6868, Y 48.8965, Z -5.5000, A 0.000, B 0.000, C 0.000 }
gfCNCPoint4[13623] = {X 302.8704, Y 48.3868, Z -5.5000, A 0.000, B 0.000, C 0.000 }
gfCNCPoint4[13624] = {X 302.1872, Y 47.7090, Z -5.5000, A 0.000, B 0.000, C 0.000 }
gfCNCPoint4[13625] = {X 301.6709, Y 46.8967, Z -5.5000, A 0.000, B 0.000, C 0.000 }
gfCNCPoint4[13626] = {X 301.3473, Y 45.9903, Z -5.5000, A 0.000, B 0.000, C 0.000 }
gfCNCPoint4[13627] = {X 301.2324, Y 45.0348, Z -5.5000, A 0.000, B 0.000, C 0.000 }
gfCNCPoint4[13628] = {X 301.2323, Y 44.2013, Z -5.5000, A 0.000, B 0.000, C 0.000 }
gfCNCPoint4[13629] = {X 301.3498, Y 43.2652, Z -5.5000, A 0.000, B 0.000, C 0.000 }
gfCNCPoint4[13630] = {X 301.6528, Y 42.3718, Z -5.5000, A 0.000, B 0.000, C 0.000 }
gfCNCPoint4[13631] = {X 302.1292, Y 41.5574, Z -5.5000, A 0.000, B 0.000, C 0.000 }
gfCNCPoint4[13632] = {X 302.7594, Y 40.8554, Z -5.5000, A 0.000, B 0.000, C 0.000 }
gfCNCPoint4[13633] = {X 302.7594, Y 34.0343, Z -5.5000, A 0.000, B 0.000, C 0.000 }
gfCNCPoint4[13634] = {X 293.8547, Y 34.0343, Z -5.5000, A 0.000, B 0.000, C 0.000 }
gfCNCPoint4[13635] = {X 293.8540, Y 40.9022, Z -5.5000, A 0.000, B 0.000, C 0.000 }
gfCNCPoint4[13636] = {X 294.4931, Y 41.5862, Z -5.5000, A 0.000, B 0.000, C 0.000 }
gfCNCPoint4[13637] = {X 294.9737, Y 42.3896, Z -5.5000, A 0.000, B 0.000, C 0.000 }
gfCNCPoint4[13638] = {X 295.2742, Y 43.2762, Z -5.5000, A 0.000, B 0.000, C 0.000 }
gfCNCPoint4[13639] = {X 295.3811, Y 44.2062, Z -5.5000, A 0.000, B 0.000, C 0.000 }
gfCNCPoint4[13640] = {X 295.3811, Y 45.0000, Z -5.5000, A 0.000, B 0.000, C 0.000 }
gfCNCPoint4[13641] = {X 295.2728, Y 45.9613, Z -5.5000, A 0.000, B 0.000, C 0.000 }
gfCNCPoint4[13642] = {X 294.9533, Y 46.8744, Z -5.5000, A 0.000, B 0.000, C 0.000 }
gfCNCPoint4[13643] = {X 294.4386, Y 47.6935, Z -5.5000, A 0.000, B 0.000, C 0.000 }
gfCNCPoint4[13644] = {X 293.7546, Y 48.3775, Z -5.5000, A 0.000, B 0.000, C 0.000 }
gfCNCPoint4[13645] = {X 292.9355, Y 48.8922, Z -5.5000, A 0.000, B 0.000, C 0.000 }
gfCNCPoint4[13646] = {X 292.0224, Y 49.2117, Z -5.5000, A 0.000, B 0.000, C 0.000 }
gfCNCPoint4[13647] = {X 291.0611, Y 49.3200, Z -5.5000, A 0.000, B 0.000, C 0.000 }
gfCNCPoint4[13648] = {X 284.6177, Y 49.3200, Z -5.5000, A 0.000, B 0.000, C 0.000 }
gfCNCPoint4[13649] = {X 283.6613, Y 49.2128, Z -5.5000, A 0.000, B 0.000, C 0.000 }
gfCNCPoint4[13650] = {X 282.7524, Y 48.8965, Z -5.5000, A 0.000, B 0.000, C 0.000 }
gfCNCPoint4[13651] = {X 281.9360, Y 48.3869, Z -5.5000, A 0.000, B 0.000, C 0.000 }
gfCNCPoint4[13652] = {X 281.2527, Y 47.7092, Z -5.5000, A 0.000, B 0.000, C 0.000 }
gfCNCPoint4[13653] = {X 280.7365, Y 46.8970, Z -5.5000, A 0.000, B 0.000, C 0.000 }
gfCNCPoint4[13654] = {X 280.4128, Y 45.9907, Z -5.5000, A 0.000, B 0.000, C 0.000 }
gfCNCPoint4[13655] = {X 280.2978, Y 45.0352, Z -5.5000, A 0.000, B 0.000, C 0.000 }
gfCNCPoint4[13656] = {X 280.2977, Y 44.2073, Z -5.5000, A 0.000, B 0.000, C 0.000 }
gfCNCPoint4[13657] = {X 280.4023, Y 43.2782, Z -5.5000, A 0.000, B 0.000, C 0.000 }
gfCNCPoint4[13658] = {X 280.7023, Y 42.3927, Z -5.5000, A 0.000, B 0.000, C 0.000 }
gfCNCPoint4[13659] = {X 281.1839, Y 41.5913, Z -5.5000, A 0.000, B 0.000, C 0.000 }
gfCNCPoint4[13660] = {X 281.8250, Y 40.9107, Z -5.5000, A 0.000, B 0.000, C 0.000 }
gfCNCPoint4[13661] = {X 281.8248, Y 28.5922, Z -5.5000, A 0.000, B 0.000, C 0.000 }
gfCNCPoint4[13662] = {X 277.8248, Y 28.5923, Z -5.5000, A 0.000, B 0.000, C 0.000 }
gfCNCPoint4[13663] = {X 281.9048, Y 28.5922, Z -5.5000, A 0.000, B 0.000, C 0.000 }
gfCNCPoint4[13664] = {X 281.9046, Y 16.2364, Z -5.5000, A 0.000, B 0.000, C 0.000 }
gfCNCPoint4[13665] = {X 281.2668, Y 15.5759, Z -5.5000, A 0.000, B 0.000, C 0.000 }
gfCNCPoint4[13666] = {X 280.7861, Y 14.7936, Z -5.5000, A 0.000, B 0.000, C 0.000 }
gfCNCPoint4[13667] = {X 280.4850, Y 13.9262, Z -5.5000, A 0.000, B 0.000, C 0.000 }
gfCNCPoint4[13668] = {X 280.3778, Y 13.0143, Z -5.5000, A 0.000, B 0.000, C 0.000 }
gfCNCPoint4[13669] = {X 280.3777, Y 12.1868, Z -5.5000, A 0.000, B 0.000, C 0.000 }
gfCNCPoint4[13670] = {X 280.4840, Y 11.2433, Z -5.5000, A 0.000, B 0.000, C 0.000 }
gfCNCPoint4[13671] = {X 280.7976, Y 10.3472, Z -5.5000, A 0.000, B 0.000, C 0.000 }
gfCNCPoint4[13672] = {X 281.3027, Y 9.5432, Z -5.5000, A 0.000, B 0.000, C 0.000 }
gfCNCPoint4[13673] = {X 281.9741, Y 8.8719, Z -5.5000, A 0.000, B 0.000, C 0.000 }
gfCNCPoint4[13674] = {X 282.7780, Y 8.3667, Z -5.5000, A 0.000, B 0.000, C 0.000 }
gfCNCPoint4[13675] = {X 283.6742, Y 8.0531, Z -5.5000, A 0.000, B 0.000, C 0.000 }
gfCNCPoint4[13676] = {X 284.6177, Y 7.9468, Z -5.5000, A 0.000, B 0.000, C 0.000 }
gfCNCPoint4[13677] = {X 291.0611, Y 7.9468, Z -5.5000, A 0.000, B 0.000, C 0.000 }
gfCNCPoint4[13678] = {X 292.0046, Y 8.0531, Z -5.5000, A 0.000, B 0.000, C 0.000 }
gfCNCPoint4[13679] = {X 292.9008, Y 8.3667, Z -5.5000, A 0.000, B 0.000, C 0.000 }
gfCNCPoint4[13680] = {X 293.7047, Y 8.8718, Z -5.5000, A 0.000, B 0.000, C 0.000 }
gfCNCPoint4[13681] = {X 294.3761, Y 9.5432, Z -5.5000, A 0.000, B 0.000, C 0.000 }
gfCNCPoint4[13682] = {X 294.8812, Y 10.3471, Z -5.5000, A 0.000, B 0.000, C 0.000 }
gfCNCPoint4[13683] = {X 295.1948, Y 11.2433, Z -5.5000, A 0.000, B 0.000, C 0.000 }
gfCNCPoint4[13684] = {X 295.3011, Y 12.1868, Z -5.5000, A 0.000, B 0.000, C 0.000 }
gfCNCPoint4[13685] = {X 295.3011, Y 12.9782, Z -5.5000, A 0.000, B 0.000, C 0.000 }
gfCNCPoint4[13686] = {X 295.1996, Y 13.8997, Z -5.5000, A 0.000, B 0.000, C 0.000 }
gfCNCPoint4[13687] = {X 294.9003, Y 14.7772, Z -5.5000, A 0.000, B 0.000, C 0.000 }
gfCNCPoint4[13688] = {X 294.4173, Y 15.5687, Z -5.5000, A 0.000, B 0.000, C 0.000 }
gfCNCPoint4[13689] = {X 293.7739, Y 16.2362, Z -5.5000, A 0.000, B 0.000, C 0.000 }
gfCNCPoint4[13690] = {X 293.7750, Y 22.2765, Z -5.5000, A 0.000, B 0.000, C 0.000 }
gfCNCPoint4[13691] = {X 302.8388, Y 22.2765, Z -5.5000, A 0.000, B 0.000, C 0.000 }
gfCNCPoint4[13692] = {X 302.8439, Y 16.2403, Z -5.5000, A 0.000, B 0.000, C 0.000 }
gfCNCPoint4[13693] = {X 302.2044, Y 15.5798, Z -5.5000, A 0.000, B 0.000, C 0.000 }
gfCNCPoint4[13694] = {X 301.7223, Y 14.7971, Z -5.5000, A 0.000, B 0.000, C 0.000 }
gfCNCPoint4[13695] = {X 301.4202, Y 13.9288, Z -5.5000, A 0.000, B 0.000, C 0.000 }
gfCNCPoint4[13696] = {X 301.3124, Y 13.0158, Z -5.5000, A 0.000, B 0.000, C 0.000 }
gfCNCPoint4[13697] = {X 301.3123, Y 12.1868, Z -5.5000, A 0.000, B 0.000, C 0.000 }
gfCNCPoint4[13698] = {X 301.4186, Y 11.2433, Z -5.5000, A 0.000, B 0.000, C 0.000 }
gfCNCPoint4[13699] = {X 301.7321, Y 10.3471, Z -5.5000, A 0.000, B 0.000, C 0.000 }
gfCNCPoint4[13700] = {X 302.2373, Y 9.5432, Z -5.5000, A 0.000, B 0.000, C 0.000 }
gfCNCPoint4[13701] = {X 302.9087, Y 8.8718, Z -5.5000, A 0.000, B 0.000, C 0.000 }
gfCNCPoint4[13702] = {X 303.7126, Y 8.3667, Z -5.5000, A 0.000, B 0.000, C 0.000 }
gfCNCPoint4[13703] = {X 304.6088, Y 8.0531, Z -5.5000, A 0.000, B 0.000, C 0.000 }
gfCNCPoint4[13704] = {X 305.5523, Y 7.9468, Z -5.5000, A 0.000, B 0.000, C 0.000 }
gfCNCPoint4[13705] = {X 311.9957, Y 7.9468, Z -5.5000, A 0.000, B 0.000, C 0.000 }
gfCNCPoint4[13706] = {X 312.9392, Y 8.0531, Z -5.5000, A 0.000, B 0.000, C 0.000 }
gfCNCPoint4[13707] = {X 313.8354, Y 8.3667, Z -5.5000, A 0.000, B 0.000, C 0.000 }
gfCNCPoint4[13708] = {X 314.6393, Y 8.8718, Z -5.5000, A 0.000, B 0.000, C 0.000 }
gfCNCPoint4[13709] = {X 315.3107, Y 9.5432, Z -5.5000, A 0.000, B 0.000, C 0.000 }
gfCNCPoint4[13710] = {X 315.8158, Y 10.3471, Z -5.5000, A 0.000, B 0.000, C 0.000 }
gfCNCPoint4[13711] = {X 316.1294, Y 11.2433, Z -5.5000, A 0.000, B 0.000, C 0.000 }
gfCNCPoint4[13712] = {X 316.2357, Y 12.1868, Z -5.5000, A 0.000, B 0.000, C 0.000 }
gfCNCPoint4[13713] = {X 316.2357, Y 12.9782, Z -5.5000, A 0.000, B 0.000, C 0.000 }
gfCNCPoint4[13714] = {X 316.1344, Y 13.8995, Z -5.5000, A 0.000, B 0.000, C 0.000 }
gfCNCPoint4[13715] = {X 315.8352, Y 14.7768, Z -5.5000, A 0.000, B 0.000, C 0.000 }
gfCNCPoint4[13716] = {X 315.3526, Y 15.5682, Z -5.5000, A 0.000, B 0.000, C 0.000 }
gfCNCPoint4[13717] = {X 314.7095, Y 16.2358, Z -5.5000, A 0.000, B 0.000, C 0.000 }
gfCNCPoint4[13718] = {X 314.7084, Y 40.9511, Z -5.5000, A 0.000, B 0.000, C 0.000 }
gfCNCPoint4[13719] = {X 314.7367, Y 40.9739, Z -5.5000, A 0.000, B 0.000, C 0.000 }
gfCNCPoint4[13720] = {X 315.3632, Y 41.6324, Z -5.5000, A 0.000, B 0.000, C 0.000 }
gfCNCPoint4[13721] = {X 315.8350, Y 42.4094, Z -5.5000, A 0.000, B 0.000, C 0.000 }
gfCNCPoint4[13722] = {X 316.1303, Y 43.2691, Z -5.5000, A 0.000, B 0.000, C 0.000 }
gfCNCPoint4[13723] = {X 316.2356, Y 44.1720, Z -5.5000, A 0.000, B 0.000, C 0.000 }
gfCNCPoint4[13724] = {X 316.2357, Y 45.0000, Z -5.5000, A 0.000, B 0.000, C 0.000 }
gfCNCPoint4[13725] = {X 316.1294, Y 45.9435, Z -5.5000, A 0.000, B 0.000, C 0.000 }
gfCNCPoint4[13726] = {X 315.8158, Y 46.8397, Z -5.5000, A 0.000, B 0.000, C 0.000 }
gfCNCPoint4[13727] = {X 315.3107, Y 47.6436, Z -5.5000, A 0.000, B 0.000, C 0.000 }
gfCNCPoint4[13728] = {X 314.6393, Y 48.3150, Z -5.5000, A 0.000, B 0.000, C 0.000 }
gfCNCPoint4[13729] = {X 313.8354, Y 48.8201, Z -5.5000, A 0.000, B 0.000, C 0.000 }
gfCNCPoint4[13730] = {X 312.9392, Y 49.1337, Z -5.5000, A 0.000, B 0.000, C 0.000 }
gfCNCPoint4[13731] = {X 311.9957, Y 49.2400, Z -5.5000, A 0.000, B 0.000, C 0.000 }
gfCNCPoint4[13732] = {X 305.5523, Y 49.2400, Z -5.5000, A 0.000, B 0.000, C 0.000 }
gfCNCPoint4[13733] = {X 304.6135, Y 49.1348, Z -5.5000, A 0.000, B 0.000, C 0.000 }
gfCNCPoint4[13734] = {X 303.7214, Y 48.8243, Z -5.5000, A 0.000, B 0.000, C 0.000 }
gfCNCPoint4[13735] = {X 302.9201, Y 48.3241, Z -5.5000, A 0.000, B 0.000, C 0.000 }
gfCNCPoint4[13736] = {X 302.2495, Y 47.6588, Z -5.5000, A 0.000, B 0.000, C 0.000 }
gfCNCPoint4[13737] = {X 301.7428, Y 46.8616, Z -5.5000, A 0.000, B 0.000, C 0.000 }
gfCNCPoint4[13738] = {X 301.4252, Y 45.9720, Z -5.5000, A 0.000, B 0.000, C 0.000 }
gfCNCPoint4[13739] = {X 301.3124, Y 45.0341, Z -5.5000, A 0.000, B 0.000, C 0.000 }
gfCNCPoint4[13740] = {X 301.3123, Y 44.2032, Z -5.5000, A 0.000, B 0.000, C 0.000 }
gfCNCPoint4[13741] = {X 301.4297, Y 43.2745, Z -5.5000, A 0.000, B 0.000, C 0.000 }
gfCNCPoint4[13742] = {X 301.7330, Y 42.3890, Z -5.5000, A 0.000, B 0.000, C 0.000 }
gfCNCPoint4[13743] = {X 302.2095, Y 41.5833, Z -5.5000, A 0.000, B 0.000, C 0.000 }
gfCNCPoint4[13744] = {X 302.8394, Y 40.8909, Z -5.5000, A 0.000, B 0.000, C 0.000 }
gfCNCPoint4[13745] = {X 302.8394, Y 33.9543, Z -5.5000, A 0.000, B 0.000, C 0.000 }
gfCNCPoint4[13746] = {X 293.7747, Y 33.9543, Z -5.5000, A 0.000, B 0.000, C 0.000 }
gfCNCPoint4[13747] = {X 293.7740, Y 40.9390, Z -5.5000, A 0.000, B 0.000, C 0.000 }
gfCNCPoint4[13748] = {X 294.4127, Y 41.6125, Z -5.5000, A 0.000, B 0.000, C 0.000 }
gfCNCPoint4[13749] = {X 294.8934, Y 42.4066, Z -5.5000, A 0.000, B 0.000, C 0.000 }
gfCNCPoint4[13750] = {X 295.1942, Y 43.2848, Z -5.5000, A 0.000, B 0.000, C 0.000 }
gfCNCPoint4[13751] = {X 295.3011, Y 44.2069, Z -5.5000, A 0.000, B 0.000, C 0.000 }
gfCNCPoint4[13752] = {X 295.3011, Y 45.0000, Z -5.5000, A 0.000, B 0.000, C 0.000 }
gfCNCPoint4[13753] = {X 295.1948, Y 45.9435, Z -5.5000, A 0.000, B 0.000, C 0.000 }
gfCNCPoint4[13754] = {X 294.8812, Y 46.8397, Z -5.5000, A 0.000, B 0.000, C 0.000 }
gfCNCPoint4[13755] = {X 294.3761, Y 47.6436, Z -5.5000, A 0.000, B 0.000, C 0.000 }
gfCNCPoint4[13756] = {X 293.7047, Y 48.3150, Z -5.5000, A 0.000, B 0.000, C 0.000 }
gfCNCPoint4[13757] = {X 292.9008, Y 48.8201, Z -5.5000, A 0.000, B 0.000, C 0.000 }
gfCNCPoint4[13758] = {X 292.0046, Y 49.1337, Z -5.5000, A 0.000, B 0.000, C 0.000 }
gfCNCPoint4[13759] = {X 291.0611, Y 49.2400, Z -5.5000, A 0.000, B 0.000, C 0.000 }
gfCNCPoint4[13760] = {X 284.6177, Y 49.2400, Z -5.5000, A 0.000, B 0.000, C 0.000 }
gfCNCPoint4[13761] = {X 283.6790, Y 49.1348, Z -5.5000, A 0.000, B 0.000, C 0.000 }
gfCNCPoint4[13762] = {X 282.7869, Y 48.8244, Z -5.5000, A 0.000, B 0.000, C 0.000 }
gfCNCPoint4[13763] = {X 281.9857, Y 48.3242, Z -5.5000, A 0.000, B 0.000, C 0.000 }
gfCNCPoint4[13764] = {X 281.3150, Y 47.6590, Z -5.5000, A 0.000, B 0.000, C 0.000 }
gfCNCPoint4[13765] = {X 280.8083, Y 46.8619, Z -5.5000, A 0.000, B 0.000, C 0.000 }
gfCNCPoint4[13766] = {X 280.4907, Y 45.9723, Z -5.5000, A 0.000, B 0.000, C 0.000 }
gfCNCPoint4[13767] = {X 280.3778, Y 45.0345, Z -5.5000, A 0.000, B 0.000, C 0.000 }
gfCNCPoint4[13768] = {X 280.3777, Y 44.2077, Z -5.5000, A 0.000, B 0.000, C 0.000 }
gfCNCPoint4[13769] = {X 280.4824, Y 43.2867, Z -5.5000, A 0.000, B 0.000, C 0.000 }
gfCNCPoint4[13770] = {X 280.7826, Y 42.4097, Z -5.5000, A 0.000, B 0.000, C 0.000 }
gfCNCPoint4[13771] = {X 281.2643, Y 41.6177, Z -5.5000, A 0.000, B 0.000, C 0.000 }
gfCNCPoint4[13772] = {X 281.9050, Y 40.9478, Z -5.5000, A 0.000, B 0.000, C 0.000 }
gfCNCPoint4[13773] = {X 281.9048, Y 28.5922, Z -5.5000, A 0.000, B 0.000, C 0.000 }
gfCNCPoint4[13774] = {X 277.9048, Y 28.5923, Z -5.5000, A 0.000, B 0.000, C 0.000 }
gfCNCPoint4[13775] = {X 281.9848, Y 28.5922, Z -5.5000, A 0.000, B 0.000, C 0.000 }
gfCNCPoint4[13776] = {X 281.9846, Y 16.1987, Z -5.5000, A 0.000, B 0.000, C 0.000 }
gfCNCPoint4[13777] = {X 281.3472, Y 15.5490, Z -5.5000, A 0.000, B 0.000, C 0.000 }
gfCNCPoint4[13778] = {X 280.8664, Y 14.7762, Z -5.5000, A 0.000, B 0.000, C 0.000 }
gfCNCPoint4[13779] = {X 280.5651, Y 13.9174, Z -5.5000, A 0.000, B 0.000, C 0.000 }
gfCNCPoint4[13780] = {X 280.4578, Y 13.0136, Z -5.5000, A 0.000, B 0.000, C 0.000 }
gfCNCPoint4[13781] = {X 280.4577, Y 12.1868, Z -5.5000, A 0.000, B 0.000, C 0.000 }
gfCNCPoint4[13782] = {X 280.5620, Y 11.2611, Z -5.5000, A 0.000, B 0.000, C 0.000 }
gfCNCPoint4[13783] = {X 280.8696, Y 10.3819, Z -5.5000, A 0.000, B 0.000, C 0.000 }
gfCNCPoint4[13784] = {X 281.3652, Y 9.5931, Z -5.5000, A 0.000, B 0.000, C 0.000 }
gfCNCPoint4[13785] = {X 282.0240, Y 8.9344, Z -5.5000, A 0.000, B 0.000, C 0.000 }
gfCNCPoint4[13786] = {X 282.8127, Y 8.4388, Z -5.5000, A 0.000, B 0.000, C 0.000 }
gfCNCPoint4[13787] = {X 283.6920, Y 8.1311, Z -5.5000, A 0.000, B 0.000, C 0.000 }
gfCNCPoint4[13788] = {X 284.6177, Y 8.0268, Z -5.5000, A 0.000, B 0.000, C 0.000 }
gfCNCPoint4[13789] = {X 291.0611, Y 8.0268, Z -5.5000, A 0.000, B 0.000, C 0.000 }
gfCNCPoint4[13790] = {X 291.9868, Y 8.1311, Z -5.5000, A 0.000, B 0.000, C 0.000 }
gfCNCPoint4[13791] = {X 292.8661, Y 8.4388, Z -5.5000, A 0.000, B 0.000, C 0.000 }
gfCNCPoint4[13792] = {X 293.6549, Y 8.9344, Z -5.5000, A 0.000, B 0.000, C 0.000 }
gfCNCPoint4[13793] = {X 294.3136, Y 9.5931, Z -5.5000, A 0.000, B 0.000, C 0.000 }
gfCNCPoint4[13794] = {X 294.8092, Y 10.3819, Z -5.5000, A 0.000, B 0.000, C 0.000 }
gfCNCPoint4[13795] = {X 295.1168, Y 11.2611, Z -5.5000, A 0.000, B 0.000, C 0.000 }
gfCNCPoint4[13796] = {X 295.2211, Y 12.1868, Z -5.5000, A 0.000, B 0.000, C 0.000 }
gfCNCPoint4[13797] = {X 295.2211, Y 12.9782, Z -5.5000, A 0.000, B 0.000, C 0.000 }
gfCNCPoint4[13798] = {X 295.1255, Y 13.8650, Z -5.5000, A 0.000, B 0.000, C 0.000 }
gfCNCPoint4[13799] = {X 294.8429, Y 14.7111, Z -5.5000, A 0.000, B 0.000, C 0.000 }
gfCNCPoint4[13800] = {X 294.3865, Y 15.4775, Z -5.5000, A 0.000, B 0.000, C 0.000 }
gfCNCPoint4[13801] = {X 293.7772, Y 16.1290, Z -5.5000, A 0.000, B 0.000, C 0.000 }
gfCNCPoint4[13802] = {X 293.6939, Y 16.1989, Z -5.5000, A 0.000, B 0.000, C 0.000 }
gfCNCPoint4[13803] = {X 293.6950, Y 22.3565, Z -5.5000, A 0.000, B 0.000, C 0.000 }
gfCNCPoint4[13804] = {X 302.9188, Y 22.3565, Z -5.5000, A 0.000, B 0.000, C 0.000 }
gfCNCPoint4[13805] = {X 302.9239, Y 16.2025, Z -5.5000, A 0.000, B 0.000, C 0.000 }
gfCNCPoint4[13806] = {X 302.2849, Y 15.5529, Z -5.5000, A 0.000, B 0.000, C 0.000 }
gfCNCPoint4[13807] = {X 301.8026, Y 14.7797, Z -5.5000, A 0.000, B 0.000, C 0.000 }
gfCNCPoint4[13808] = {X 301.5003, Y 13.9200, Z -5.5000, A 0.000, B 0.000, C 0.000 }
gfCNCPoint4[13809] = {X 301.3924, Y 13.0151, Z -5.5000, A 0.000, B 0.000, C 0.000 }
gfCNCPoint4[13810] = {X 301.3923, Y 12.1868, Z -5.5000, A 0.000, B 0.000, C 0.000 }
gfCNCPoint4[13811] = {X 301.4966, Y 11.2611, Z -5.5000, A 0.000, B 0.000, C 0.000 }
gfCNCPoint4[13812] = {X 301.8042, Y 10.3819, Z -5.5000, A 0.000, B 0.000, C 0.000 }
gfCNCPoint4[13813] = {X 302.2998, Y 9.5931, Z -5.5000, A 0.000, B 0.000, C 0.000 }
gfCNCPoint4[13814] = {X 302.9585, Y 8.9344, Z -5.5000, A 0.000, B 0.000, C 0.000 }
gfCNCPoint4[13815] = {X 303.7473, Y 8.4388, Z -5.5000, A 0.000, B 0.000, C 0.000 }
gfCNCPoint4[13816] = {X 304.6266, Y 8.1311, Z -5.5000, A 0.000, B 0.000, C 0.000 }
gfCNCPoint4[13817] = {X 305.5523, Y 8.0268, Z -5.5000, A 0.000, B 0.000, C 0.000 }
gfCNCPoint4[13818] = {X 311.9957, Y 8.0268, Z -5.5000, A 0.000, B 0.000, C 0.000 }
gfCNCPoint4[13819] = {X 312.9214, Y 8.1311, Z -5.5000, A 0.000, B 0.000, C 0.000 }
gfCNCPoint4[13820] = {X 313.8007, Y 8.4388, Z -5.5000, A 0.000, B 0.000, C 0.000 }
gfCNCPoint4[13821] = {X 314.5894, Y 8.9344, Z -5.5000, A 0.000, B 0.000, C 0.000 }
gfCNCPoint4[13822] = {X 315.2481, Y 9.5931, Z -5.5000, A 0.000, B 0.000, C 0.000 }
gfCNCPoint4[13823] = {X 315.7438, Y 10.3819, Z -5.5000, A 0.000, B 0.000, C 0.000 }
gfCNCPoint4[13824] = {X 316.0514, Y 11.2611, Z -5.5000, A 0.000, B 0.000, C 0.000 }
gfCNCPoint4[13825] = {X 316.1557, Y 12.1868, Z -5.5000, A 0.000, B 0.000, C 0.000 }
gfCNCPoint4[13826] = {X 316.1557, Y 12.9782, Z -5.5000, A 0.000, B 0.000, C 0.000 }
gfCNCPoint4[13827] = {X 316.0542, Y 13.8912, Z -5.5000, A 0.000, B 0.000, C 0.000 }
gfCNCPoint4[13828] = {X 315.7548, Y 14.7598, Z -5.5000, A 0.000, B 0.000, C 0.000 }
gfCNCPoint4[13829] = {X 315.2721, Y 15.5414, Z -5.5000, A 0.000, B 0.000, C 0.000 }
gfCNCPoint4[13830] = {X 314.6295, Y 16.1981, Z -5.5000, A 0.000, B 0.000, C 0.000 }
gfCNCPoint4[13831] = {X 314.6284, Y 40.9895, Z -5.5000, A 0.000, B 0.000, C 0.000 }
gfCNCPoint4[13832] = {X 314.6836, Y 41.0338, Z -5.5000, A 0.000, B 0.000, C 0.000 }
gfCNCPoint4[13833] = {X 315.2989, Y 41.6800, Z -5.5000, A 0.000, B 0.000, C 0.000 }
gfCNCPoint4[13834] = {X 315.7622, Y 42.4426, Z -5.5000, A 0.000, B 0.000, C 0.000 }
gfCNCPoint4[13835] = {X 316.0522, Y 43.2864, Z -5.5000, A 0.000, B 0.000, C 0.000 }
gfCNCPoint4[13836] = {X 316.1556, Y 44.1727, Z -5.5000, A 0.000, B 0.000, C 0.000 }
gfCNCPoint4[13837] = {X 316.1557, Y 45.0000, Z -5.5000, A 0.000, B 0.000, C 0.000 }
gfCNCPoint4[13838] = {X 316.0514, Y 45.9257, Z -5.5000, A 0.000, B 0.000, C 0.000 }
gfCNCPoint4[13839] = {X 315.7438, Y 46.8050, Z -5.5000, A 0.000, B 0.000, C 0.000 }
gfCNCPoint4[13840] = {X 315.2481, Y 47.5937, Z -5.5000, A 0.000, B 0.000, C 0.000 }
gfCNCPoint4[13841] = {X 314.5894, Y 48.2524, Z -5.5000, A 0.000, B 0.000, C 0.000 }
gfCNCPoint4[13842] = {X 313.8007, Y 48.7480, Z -5.5000, A 0.000, B 0.000, C 0.000 }
gfCNCPoint4[13843] = {X 312.9214, Y 49.0557, Z -5.5000, A 0.000, B 0.000, C 0.000 }
gfCNCPoint4[13844] = {X 311.9957, Y 49.1600, Z -5.5000, A 0.000, B 0.000, C 0.000 }
gfCNCPoint4[13845] = {X 305.5523, Y 49.1600, Z -5.5000, A 0.000, B 0.000, C 0.000 }
gfCNCPoint4[13846] = {X 304.6312, Y 49.0568, Z -5.5000, A 0.000, B 0.000, C 0.000 }
gfCNCPoint4[13847] = {X 303.7559, Y 48.7522, Z -5.5000, A 0.000, B 0.000, C 0.000 }
gfCNCPoint4[13848] = {X 302.9698, Y 48.2613, Z -5.5000, A 0.000, B 0.000, C 0.000 }
gfCNCPoint4[13849] = {X 302.3118, Y 47.6087, Z -5.5000, A 0.000, B 0.000, C 0.000 }
gfCNCPoint4[13850] = {X 301.8147, Y 46.8265, Z -5.5000, A 0.000, B 0.000, C 0.000 }
gfCNCPoint4[13851] = {X 301.5030, Y 45.9537, Z -5.5000, A 0.000, B 0.000, C 0.000 }
gfCNCPoint4[13852] = {X 301.3924, Y 45.0335, Z -5.5000, A 0.000, B 0.000, C 0.000 }
gfCNCPoint4[13853] = {X 301.3923, Y 44.2051, Z -5.5000, A 0.000, B 0.000, C 0.000 }
gfCNCPoint4[13854] = {X 301.5097, Y 43.2839, Z -5.5000, A 0.000, B 0.000, C 0.000 }
gfCNCPoint4[13855] = {X 301.8131, Y 42.4063, Z -5.5000, A 0.000, B 0.000, C 0.000 }
gfCNCPoint4[13856] = {X 302.2897, Y 41.6094, Z -5.5000, A 0.000, B 0.000, C 0.000 }
gfCNCPoint4[13857] = {X 302.9194, Y 40.9268, Z -5.5000, A 0.000, B 0.000, C 0.000 }
gfCNCPoint4[13858] = {X 302.9194, Y 33.8743, Z -5.5000, A 0.000, B 0.000, C 0.000 }
gfCNCPoint4[13859] = {X 293.6947, Y 33.8743, Z -5.5000, A 0.000, B 0.000, C 0.000 }
gfCNCPoint4[13860] = {X 293.6940, Y 40.9762, Z -5.5000, A 0.000, B 0.000, C 0.000 }
gfCNCPoint4[13861] = {X 294.3322, Y 41.6391, Z -5.5000, A 0.000, B 0.000, C 0.000 }
gfCNCPoint4[13862] = {X 294.8131, Y 42.4238, Z -5.5000, A 0.000, B 0.000, C 0.000 }
gfCNCPoint4[13863] = {X 295.1141, Y 43.2935, Z -5.5000, A 0.000, B 0.000, C 0.000 }
gfCNCPoint4[13864] = {X 295.2211, Y 44.2076, Z -5.5000, A 0.000, B 0.000, C 0.000 }
gfCNCPoint4[13865] = {X 295.2211, Y 45.0000, Z -5.5000, A 0.000, B 0.000, C 0.000 }
gfCNCPoint4[13866] = {X 295.1168, Y 45.9257, Z -5.5000, A 0.000, B 0.000, C 0.000 }
gfCNCPoint4[13867] = {X 294.8092, Y 46.8050, Z -5.5000, A 0.000, B 0.000, C 0.000 }
gfCNCPoint4[13868] = {X 294.3136, Y 47.5937, Z -5.5000, A 0.000, B 0.000, C 0.000 }
gfCNCPoint4[13869] = {X 293.6549, Y 48.2524, Z -5.5000, A 0.000, B 0.000, C 0.000 }
gfCNCPoint4[13870] = {X 292.8661, Y 48.7480, Z -5.5000, A 0.000, B 0.000, C 0.000 }
gfCNCPoint4[13871] = {X 291.9868, Y 49.0557, Z -5.5000, A 0.000, B 0.000, C 0.000 }
gfCNCPoint4[13872] = {X 291.0611, Y 49.1600, Z -5.5000, A 0.000, B 0.000, C 0.000 }
gfCNCPoint4[13873] = {X 284.6177, Y 49.1600, Z -5.5000, A 0.000, B 0.000, C 0.000 }
gfCNCPoint4[13874] = {X 283.6967, Y 49.0568, Z -5.5000, A 0.000, B 0.000, C 0.000 }
gfCNCPoint4[13875] = {X 282.8214, Y 48.7522, Z -5.5000, A 0.000, B 0.000, C 0.000 }
gfCNCPoint4[13876] = {X 282.0353, Y 48.2615, Z -5.5000, A 0.000, B 0.000, C 0.000 }
gfCNCPoint4[13877] = {X 281.3774, Y 47.6088, Z -5.5000, A 0.000, B 0.000, C 0.000 }
gfCNCPoint4[13878] = {X 280.8802, Y 46.8267, Z -5.5000, A 0.000, B 0.000, C 0.000 }
gfCNCPoint4[13879] = {X 280.5685, Y 45.9540, Z -5.5000, A 0.000, B 0.000, C 0.000 }
gfCNCPoint4[13880] = {X 280.4578, Y 45.0339, Z -5.5000, A 0.000, B 0.000, C 0.000 }
gfCNCPoint4[13881] = {X 280.4577, Y 44.2081, Z -5.5000, A 0.000, B 0.000, C 0.000 }
gfCNCPoint4[13882] = {X 280.5625, Y 43.2952, Z -5.5000, A 0.000, B 0.000, C 0.000 }
gfCNCPoint4[13883] = {X 280.8630, Y 42.4268, Z -5.5000, A 0.000, B 0.000, C 0.000 }
gfCNCPoint4[13884] = {X 281.3448, Y 41.6444, Z -5.5000, A 0.000, B 0.000, C 0.000 }
gfCNCPoint4[13885] = {X 281.9850, Y 40.9852, Z -5.5000, A 0.000, B 0.000, C 0.000 }
gfCNCPoint4[13886] = {X 281.9848, Y 28.5922, Z -5.5000, A 0.000, B 0.000, C 0.000 }
gfCNCPoint4[13887] = {X 277.9848, Y 28.5923, Z -5.5000, A 0.000, B 0.000, C 0.000 }
gfCNCPoint4[13888] = {X 282.0648, Y 28.5922, Z -5.5000, A 0.000, B 0.000, C 0.000 }
gfCNCPoint4[13889] = {X 282.0646, Y 16.1605, Z -5.5000, A 0.000, B 0.000, C 0.000 }
gfCNCPoint4[13890] = {X 281.4277, Y 15.5218, Z -5.5000, A 0.000, B 0.000, C 0.000 }
gfCNCPoint4[13891] = {X 280.9467, Y 14.7587, Z -5.5000, A 0.000, B 0.000, C 0.000 }
gfCNCPoint4[13892] = {X 280.6452, Y 13.9085, Z -5.5000, A 0.000, B 0.000, C 0.000 }
gfCNCPoint4[13893] = {X 280.5378, Y 13.0129, Z -5.5000, A 0.000, B 0.000, C 0.000 }
gfCNCPoint4[13894] = {X 280.5377, Y 12.1868, Z -5.5000, A 0.000, B 0.000, C 0.000 }
gfCNCPoint4[13895] = {X 280.6400, Y 11.2789, Z -5.5000, A 0.000, B 0.000, C 0.000 }
gfCNCPoint4[13896] = {X 280.9417, Y 10.4166, Z -5.5000, A 0.000, B 0.000, C 0.000 }
gfCNCPoint4[13897] = {X 281.4278, Y 9.6430, Z -5.5000, A 0.000, B 0.000, C 0.000 }
gfCNCPoint4[13898] = {X 282.0738, Y 8.9969, Z -5.5000, A 0.000, B 0.000, C 0.000 }
gfCNCPoint4[13899] = {X 282.8474, Y 8.5109, Z -5.5000, A 0.000, B 0.000, C 0.000 }
gfCNCPoint4[13900] = {X 283.7098, Y 8.2091, Z -5.5000, A 0.000, B 0.000, C 0.000 }
gfCNCPoint4[13901] = {X 284.6177, Y 8.1068, Z -5.5000, A 0.000, B 0.000, C 0.000 }
gfCNCPoint4[13902] = {X 291.0611, Y 8.1068, Z -5.5000, A 0.000, B 0.000, C 0.000 }
gfCNCPoint4[13903] = {X 291.9690, Y 8.2091, Z -5.5000, A 0.000, B 0.000, C 0.000 }
gfCNCPoint4[13904] = {X 292.8314, Y 8.5109, Z -5.5000, A 0.000, B 0.000, C 0.000 }
gfCNCPoint4[13905] = {X 293.6050, Y 8.9969, Z -5.5000, A 0.000, B 0.000, C 0.000 }
gfCNCPoint4[13906] = {X 294.2510, Y 9.6430, Z -5.5000, A 0.000, B 0.000, C 0.000 }
gfCNCPoint4[13907] = {X 294.7371, Y 10.4166, Z -5.5000, A 0.000, B 0.000, C 0.000 }
gfCNCPoint4[13908] = {X 295.0388, Y 11.2789, Z -5.5000, A 0.000, B 0.000, C 0.000 }
gfCNCPoint4[13909] = {X 295.1411, Y 12.1868, Z -5.5000, A 0.000, B 0.000, C 0.000 }
gfCNCPoint4[13910] = {X 295.1411, Y 12.9782, Z -5.5000, A 0.000, B 0.000, C 0.000 }
gfCNCPoint4[13911] = {X 295.0473, Y 13.8480, Z -5.5000, A 0.000, B 0.000, C 0.000 }
gfCNCPoint4[13912] = {X 294.7702, Y 14.6778, Z -5.5000, A 0.000, B 0.000, C 0.000 }
gfCNCPoint4[13913] = {X 294.3226, Y 15.4295, Z -5.5000, A 0.000, B 0.000, C 0.000 }
gfCNCPoint4[13914] = {X 293.7250, Y 16.0684, Z -5.5000, A 0.000, B 0.000, C 0.000 }
gfCNCPoint4[13915] = {X 293.6675, Y 16.1170, Z -5.5000, A 0.000, B 0.000, C 0.000 }
gfCNCPoint4[13916] = {X 293.6091, Y 16.1646, Z -5.5000, A 0.000, B 0.000, C 0.000 }
gfCNCPoint4[13917] = {X 293.6139, Y 16.1990, Z -5.5000, A 0.000, B 0.000, C 0.000 }
gfCNCPoint4[13918] = {X 293.6150, Y 22.4365, Z -5.5000, A 0.000, B 0.000, C 0.000 }
gfCNCPoint4[13919] = {X 302.9987, Y 22.4365, Z -5.5000, A 0.000, B 0.000, C 0.000 }
gfCNCPoint4[13920] = {X 303.0040, Y 16.1643, Z -5.5000, A 0.000, B 0.000, C 0.000 }
gfCNCPoint4[13921] = {X 302.9456, Y 16.1167, Z -5.5000, A 0.000, B 0.000, C 0.000 }
gfCNCPoint4[13922] = {X 302.8881, Y 16.0681, Z -5.5000, A 0.000, B 0.000, C 0.000 }
gfCNCPoint4[13923] = {X 302.2961, Y 15.4364, Z -5.5000, A 0.000, B 0.000, C 0.000 }
gfCNCPoint4[13924] = {X 301.8507, Y 14.6940, Z -5.5000, A 0.000, B 0.000, C 0.000 }
gfCNCPoint4[13925] = {X 301.5719, Y 13.8744, Z -5.5000, A 0.000, B 0.000, C 0.000 }
gfCNCPoint4[13926] = {X 301.4724, Y 13.0144, Z -5.5000, A 0.000, B 0.000, C 0.000 }
gfCNCPoint4[13927] = {X 301.4723, Y 12.1868, Z -5.5000, A 0.000, B 0.000, C 0.000 }
gfCNCPoint4[13928] = {X 301.5745, Y 11.2789, Z -5.5000, A 0.000, B 0.000, C 0.000 }
gfCNCPoint4[13929] = {X 301.8763, Y 10.4166, Z -5.5000, A 0.000, B 0.000, C 0.000 }
gfCNCPoint4[13930] = {X 302.3624, Y 9.6430, Z -5.5000, A 0.000, B 0.000, C 0.000 }
gfCNCPoint4[13931] = {X 303.0084, Y 8.9969, Z -5.5000, A 0.000, B 0.000, C 0.000 }
gfCNCPoint4[13932] = {X 303.7820, Y 8.5109, Z -5.5000, A 0.000, B 0.000, C 0.000 }
gfCNCPoint4[13933] = {X 304.6444, Y 8.2091, Z -5.5000, A 0.000, B 0.000, C 0.000 }
gfCNCPoint4[13934] = {X 305.5523, Y 8.1068, Z -5.5000, A 0.000, B 0.000, C 0.000 }
gfCNCPoint4[13935] = {X 311.9957, Y 8.1068, Z -5.5000, A 0.000, B 0.000, C 0.000 }
gfCNCPoint4[13936] = {X 312.9036, Y 8.2091, Z -5.5000, A 0.000, B 0.000, C 0.000 }
gfCNCPoint4[13937] = {X 313.7660, Y 8.5109, Z -5.5000, A 0.000, B 0.000, C 0.000 }
gfCNCPoint4[13938] = {X 314.5396, Y 8.9969, Z -5.5000, A 0.000, B 0.000, C 0.000 }
gfCNCPoint4[13939] = {X 315.1856, Y 9.6430, Z -5.5000, A 0.000, B 0.000, C 0.000 }
gfCNCPoint4[13940] = {X 315.6717, Y 10.4166, Z -5.5000, A 0.000, B 0.000, C 0.000 }
gfCNCPoint4[13941] = {X 315.9734, Y 11.2789, Z -5.5000, A 0.000, B 0.000, C 0.000 }
gfCNCPoint4[13942] = {X 316.0757, Y 12.1868, Z -5.5000, A 0.000, B 0.000, C 0.000 }
gfCNCPoint4[13943] = {X 316.0757, Y 12.9782, Z -5.5000, A 0.000, B 0.000, C 0.000 }
gfCNCPoint4[13944] = {X 315.9741, Y 13.8829, Z -5.5000, A 0.000, B 0.000, C 0.000 }
gfCNCPoint4[13945] = {X 315.6744, Y 14.7426, Z -5.5000, A 0.000, B 0.000, C 0.000 }
gfCNCPoint4[13946] = {X 315.1915, Y 15.5144, Z -5.5000, A 0.000, B 0.000, C 0.000 }
gfCNCPoint4[13947] = {X 314.5495, Y 16.1599, Z -5.5000, A 0.000, B 0.000, C 0.000 }
gfCNCPoint4[13948] = {X 314.5484, Y 41.0279, Z -5.5000, A 0.000, B 0.000, C 0.000 }
gfCNCPoint4[13949] = {X 314.6336, Y 41.0962, Z -5.5000, A 0.000, B 0.000, C 0.000 }
gfCNCPoint4[13950] = {X 315.2363, Y 41.7299, Z -5.5000, A 0.000, B 0.000, C 0.000 }
gfCNCPoint4[13951] = {X 315.6902, Y 42.4775, Z -5.5000, A 0.000, B 0.000, C 0.000 }
gfCNCPoint4[13952] = {X 315.9743, Y 43.3047, Z -5.5000, A 0.000, B 0.000, C 0.000 }
gfCNCPoint4[13953] = {X 316.0756, Y 44.1734, Z -5.5000, A 0.000, B 0.000, C 0.000 }
gfCNCPoint4[13954] = {X 316.0757, Y 45.0000, Z -5.5000, A 0.000, B 0.000, C 0.000 }
gfCNCPoint4[13955] = {X 315.9734, Y 45.9079, Z -5.5000, A 0.000, B 0.000, C 0.000 }
gfCNCPoint4[13956] = {X 315.6717, Y 46.7702, Z -5.5000, A 0.000, B 0.000, C 0.000 }
gfCNCPoint4[13957] = {X 315.1856, Y 47.5438, Z -5.5000, A 0.000, B 0.000, C 0.000 }
gfCNCPoint4[13958] = {X 314.5396, Y 48.1899, Z -5.5000, A 0.000, B 0.000, C 0.000 }
gfCNCPoint4[13959] = {X 313.7660, Y 48.6760, Z -5.5000, A 0.000, B 0.000, C 0.000 }
gfCNCPoint4[13960] = {X 312.9036, Y 48.9777, Z -5.5000, A 0.000, B 0.000, C 0.000 }
gfCNCPoint4[13961] = {X 311.9957, Y 49.0800, Z -5.5000, A 0.000, B 0.000, C 0.000 }
gfCNCPoint4[13962] = {X 305.5523, Y 49.0800, Z -5.5000, A 0.000, B 0.000, C 0.000 }
gfCNCPoint4[13963] = {X 304.6489, Y 48.9787, Z -5.5000, A 0.000, B 0.000, C 0.000 }
gfCNCPoint4[13964] = {X 303.7905, Y 48.6800, Z -5.5000, A 0.000, B 0.000, C 0.000 }
gfCNCPoint4[13965] = {X 303.0194, Y 48.1986, Z -5.5000, A 0.000, B 0.000, C 0.000 }
gfCNCPoint4[13966] = {X 302.3741, Y 47.5585, Z -5.5000, A 0.000, B 0.000, C 0.000 }
gfCNCPoint4[13967] = {X 301.8865, Y 46.7914, Z -5.5000, A 0.000, B 0.000, C 0.000 }
gfCNCPoint4[13968] = {X 301.5809, Y 45.9353, Z -5.5000, A 0.000, B 0.000, C 0.000 }
gfCNCPoint4[13969] = {X 301.4724, Y 45.0328, Z -5.5000, A 0.000, B 0.000, C 0.000 }
gfCNCPoint4[13970] = {X 301.4723, Y 44.2070, Z -5.5000, A 0.000, B 0.000, C 0.000 }
gfCNCPoint4[13971] = {X 301.5896, Y 43.2934, Z -5.5000, A 0.000, B 0.000, C 0.000 }
gfCNCPoint4[13972] = {X 301.8933, Y 42.4238, Z -5.5000, A 0.000, B 0.000, C 0.000 }
gfCNCPoint4[13973] = {X 302.3700, Y 41.6357, Z -5.5000, A 0.000, B 0.000, C 0.000 }
gfCNCPoint4[13974] = {X 302.9994, Y 40.9632, Z -5.5000, A 0.000, B 0.000, C 0.000 }
gfCNCPoint4[13975] = {X 302.9994, Y 33.7943, Z -5.5000, A 0.000, B 0.000, C 0.000 }
gfCNCPoint4[13976] = {X 293.6147, Y 33.7943, Z -5.5000, A 0.000, B 0.000, C 0.000 }
gfCNCPoint4[13977] = {X 293.6140, Y 41.0138, Z -5.5000, A 0.000, B 0.000, C 0.000 }
gfCNCPoint4[13978] = {X 294.2518, Y 41.6660, Z -5.5000, A 0.000, B 0.000, C 0.000 }
gfCNCPoint4[13979] = {X 294.7328, Y 42.4412, Z -5.5000, A 0.000, B 0.000, C 0.000 }
gfCNCPoint4[13980] = {X 295.0340, Y 43.3023, Z -5.5000, A 0.000, B 0.000, C 0.000 }
gfCNCPoint4[13981] = {X 295.1411, Y 44.2082, Z -5.5000, A 0.000, B 0.000, C 0.000 }
gfCNCPoint4[13982] = {X 295.1411, Y 45.0000, Z -5.5000, A 0.000, B 0.000, C 0.000 }
gfCNCPoint4[13983] = {X 295.0388, Y 45.9079, Z -5.5000, A 0.000, B 0.000, C 0.000 }
gfCNCPoint4[13984] = {X 294.7371, Y 46.7702, Z -5.5000, A 0.000, B 0.000, C 0.000 }
gfCNCPoint4[13985] = {X 294.2510, Y 47.5438, Z -5.5000, A 0.000, B 0.000, C 0.000 }
gfCNCPoint4[13986] = {X 293.6050, Y 48.1899, Z -5.5000, A 0.000, B 0.000, C 0.000 }
gfCNCPoint4[13987] = {X 292.8314, Y 48.6760, Z -5.5000, A 0.000, B 0.000, C 0.000 }
gfCNCPoint4[13988] = {X 291.9690, Y 48.9777, Z -5.5000, A 0.000, B 0.000, C 0.000 }
gfCNCPoint4[13989] = {X 291.0611, Y 49.0800, Z -5.5000, A 0.000, B 0.000, C 0.000 }
gfCNCPoint4[13990] = {X 284.6177, Y 49.0800, Z -5.5000, A 0.000, B 0.000, C 0.000 }
gfCNCPoint4[13991] = {X 283.7144, Y 48.9788, Z -5.5000, A 0.000, B 0.000, C 0.000 }
gfCNCPoint4[13992] = {X 282.8560, Y 48.6801, Z -5.5000, A 0.000, B 0.000, C 0.000 }
gfCNCPoint4[13993] = {X 282.0850, Y 48.1987, Z -5.5000, A 0.000, B 0.000, C 0.000 }
gfCNCPoint4[13994] = {X 281.4397, Y 47.5587, Z -5.5000, A 0.000, B 0.000, C 0.000 }
gfCNCPoint4[13995] = {X 280.9521, Y 46.7916, Z -5.5000, A 0.000, B 0.000, C 0.000 }
gfCNCPoint4[13996] = {X 280.6464, Y 45.9356, Z -5.5000, A 0.000, B 0.000, C 0.000 }
gfCNCPoint4[13997] = {X 280.5378, Y 45.0332, Z -5.5000, A 0.000, B 0.000, C 0.000 }
gfCNCPoint4[13998] = {X 280.5377, Y 44.2085, Z -5.5000, A 0.000, B 0.000, C 0.000 }
gfCNCPoint4[13999] = {X 280.6426, Y 43.3038, Z -5.5000, A 0.000, B 0.000, C 0.000 }
gfCNCPoint4[14000] = {X 280.9433, Y 42.4441, Z -5.5000, A 0.000, B 0.000, C 0.000 }
gfCNCPoint4[14001] = {X 281.4253, Y 41.6714, Z -5.5000, A 0.000, B 0.000, C 0.000 }
gfCNCPoint4[14002] = {X 282.0650, Y 41.0231, Z -5.5000, A 0.000, B 0.000, C 0.000 }
gfCNCPoint4[14003] = {X 282.0648, Y 28.5922, Z -5.5000, A 0.000, B 0.000, C 0.000 }
gfCNCPoint4[14004] = {X 278.0648, Y 28.5923, Z -5.5000, A 0.000, B 0.000, C 0.000 }
gfCNCPoint4[14005] = {X 282.1448, Y 28.5922, Z -5.5000, A 0.000, B 0.000, C 0.000 }
gfCNCPoint4[14006] = {X 282.1446, Y 16.1219, Z -5.5000, A 0.000, B 0.000, C 0.000 }
gfCNCPoint4[14007] = {X 281.5028, Y 15.4876, Z -5.5000, A 0.000, B 0.000, C 0.000 }
gfCNCPoint4[14008] = {X 281.0196, Y 14.7255, Z -5.5000, A 0.000, B 0.000, C 0.000 }
gfCNCPoint4[14009] = {X 280.7194, Y 13.8745, Z -5.5000, A 0.000, B 0.000, C 0.000 }
gfCNCPoint4[14010] = {X 280.6177, Y 12.9780, Z -5.5000, A 0.000, B 0.000, C 0.000 }
gfCNCPoint4[14011] = {X 280.6177, Y 12.1868, Z -5.5000, A 0.000, B 0.000, C 0.000 }
gfCNCPoint4[14012] = {X 280.7180, Y 11.2967, Z -5.5000, A 0.000, B 0.000, C 0.000 }
gfCNCPoint4[14013] = {X 281.0138, Y 10.4513, Z -5.5000, A 0.000, B 0.000, C 0.000 }
gfCNCPoint4[14014] = {X 281.4903, Y 9.6929, Z -5.5000, A 0.000, B 0.000, C 0.000 }
gfCNCPoint4[14015] = {X 282.1237, Y 9.0595, Z -5.5000, A 0.000, B 0.000, C 0.000 }
gfCNCPoint4[14016] = {X 282.8821, Y 8.5829, Z -5.5000, A 0.000, B 0.000, C 0.000 }
gfCNCPoint4[14017] = {X 283.7276, Y 8.2871, Z -5.5000, A 0.000, B 0.000, C 0.000 }
gfCNCPoint4[14018] = {X 284.6177, Y 8.1868, Z -5.5000, A 0.000, B 0.000, C 0.000 }
gfCNCPoint4[14019] = {X 291.0611, Y 8.1868, Z -5.5000, A 0.000, B 0.000, C 0.000 }
gfCNCPoint4[14020] = {X 291.9512, Y 8.2871, Z -5.5000, A 0.000, B 0.000, C 0.000 }
gfCNCPoint4[14021] = {X 292.7967, Y 8.5829, Z -5.5000, A 0.000, B 0.000, C 0.000 }
gfCNCPoint4[14022] = {X 293.5551, Y 9.0595, Z -5.5000, A 0.000, B 0.000, C 0.000 }
gfCNCPoint4[14023] = {X 294.1885, Y 9.6929, Z -5.5000, A 0.000, B 0.000, C 0.000 }
gfCNCPoint4[14024] = {X 294.6650, Y 10.4513, Z -5.5000, A 0.000, B 0.000, C 0.000 }
gfCNCPoint4[14025] = {X 294.9608, Y 11.2967, Z -5.5000, A 0.000, B 0.000, C 0.000 }
gfCNCPoint4[14026] = {X 295.0611, Y 12.1868, Z -5.5000, A 0.000, B 0.000, C 0.000 }
gfCNCPoint4[14027] = {X 295.0609, Y 13.0192, Z -5.5000, A 0.000, B 0.000, C 0.000 }
gfCNCPoint4[14028] = {X 294.9625, Y 13.8610, Z -5.5000, A 0.000, B 0.000, C 0.000 }
gfCNCPoint4[14029] = {X 294.6889, Y 14.6631, Z -5.5000, A 0.000, B 0.000, C 0.000 }
gfCNCPoint4[14030] = {X 294.2524, Y 15.3896, Z -5.5000, A 0.000, B 0.000, C 0.000 }
gfCNCPoint4[14031] = {X 293.6727, Y 16.0078, Z -5.5000, A 0.000, B 0.000, C 0.000 }
gfCNCPoint4[14032] = {X 293.5960, Y 16.0723, Z -5.5000, A 0.000, B 0.000, C 0.000 }
gfCNCPoint4[14033] = {X 293.5177, Y 16.1348, Z -5.5000, A 0.000, B 0.000, C 0.000 }
gfCNCPoint4[14034] = {X 293.5339, Y 16.1925, Z -5.5000, A 0.000, B 0.000, C 0.000 }
gfCNCPoint4[14035] = {X 293.5350, Y 22.5165, Z -5.5000, A 0.000, B 0.000, C 0.000 }
gfCNCPoint4[14036] = {X 302.6787, Y 22.5165, Z -5.5000, A 0.000, B 0.000, C 0.000 }
gfCNCPoint4[14037] = {X 303.0787, Y 22.5168, Z -5.5000, A 0.000, B 0.000, C 0.000 }
gfCNCPoint4[14038] = {X 303.0791, Y 16.1926, Z -5.5000, A 0.000, B 0.000, C 0.000 }
gfCNCPoint4[14039] = {X 303.0955, Y 16.1346, Z -5.5000, A 0.000, B 0.000, C 0.000 }
gfCNCPoint4[14040] = {X 303.0171, Y 16.0720, Z -5.5000, A 0.000, B 0.000, C 0.000 }
gfCNCPoint4[14041] = {X 302.9403, Y 16.0075, Z -5.5000, A 0.000, B 0.000, C 0.000 }
gfCNCPoint4[14042] = {X 302.3545, Y 15.3811, Z -5.5000, A 0.000, B 0.000, C 0.000 }
gfCNCPoint4[14043] = {X 301.9158, Y 14.6441, Z -5.5000, A 0.000, B 0.000, C 0.000 }
gfCNCPoint4[14044] = {X 301.6442, Y 13.8306, Z -5.5000, A 0.000, B 0.000, C 0.000 }
gfCNCPoint4[14045] = {X 301.5523, Y 12.9779, Z -5.5000, A 0.000, B 0.000, C 0.000 }
gfCNCPoint4[14046] = {X 301.5523, Y 12.1868, Z -5.5000, A 0.000, B 0.000, C 0.000 }
gfCNCPoint4[14047] = {X 301.6525, Y 11.2967, Z -5.5000, A 0.000, B 0.000, C 0.000 }
gfCNCPoint4[14048] = {X 301.9484, Y 10.4513, Z -5.5000, A 0.000, B 0.000, C 0.000 }
gfCNCPoint4[14049] = {X 302.4249, Y 9.6929, Z -5.5000, A 0.000, B 0.000, C 0.000 }
gfCNCPoint4[14050] = {X 303.0583, Y 9.0595, Z -5.5000, A 0.000, B 0.000, C 0.000 }
gfCNCPoint4[14051] = {X 303.8167, Y 8.5829, Z -5.5000, A 0.000, B 0.000, C 0.000 }
gfCNCPoint4[14052] = {X 304.6622, Y 8.2871, Z -5.5000, A 0.000, B 0.000, C 0.000 }
gfCNCPoint4[14053] = {X 305.5523, Y 8.1868, Z -5.5000, A 0.000, B 0.000, C 0.000 }
gfCNCPoint4[14054] = {X 311.9957, Y 8.1868, Z -5.5000, A 0.000, B 0.000, C 0.000 }
gfCNCPoint4[14055] = {X 312.8858, Y 8.2871, Z -5.5000, A 0.000, B 0.000, C 0.000 }
gfCNCPoint4[14056] = {X 313.7313, Y 8.5829, Z -5.5000, A 0.000, B 0.000, C 0.000 }
gfCNCPoint4[14057] = {X 314.4897, Y 9.0595, Z -5.5000, A 0.000, B 0.000, C 0.000 }
gfCNCPoint4[14058] = {X 315.1230, Y 9.6929, Z -5.5000, A 0.000, B 0.000, C 0.000 }
gfCNCPoint4[14059] = {X 315.5996, Y 10.4513, Z -5.5000, A 0.000, B 0.000, C 0.000 }
gfCNCPoint4[14060] = {X 315.8954, Y 11.2967, Z -5.5000, A 0.000, B 0.000, C 0.000 }
gfCNCPoint4[14061] = {X 315.9957, Y 12.1868, Z -5.5000, A 0.000, B 0.000, C 0.000 }
gfCNCPoint4[14062] = {X 315.9955, Y 13.0192, Z -5.5000, A 0.000, B 0.000, C 0.000 }
gfCNCPoint4[14063] = {X 315.8870, Y 13.9044, Z -5.5000, A 0.000, B 0.000, C 0.000 }
gfCNCPoint4[14064] = {X 315.5850, Y 14.7436, Z -5.5000, A 0.000, B 0.000, C 0.000 }
gfCNCPoint4[14065] = {X 315.1045, Y 15.4950, Z -5.5000, A 0.000, B 0.000, C 0.000 }
gfCNCPoint4[14066] = {X 314.4695, Y 16.1213, Z -5.5000, A 0.000, B 0.000, C 0.000 }
gfCNCPoint4[14067] = {X 314.4684, Y 41.0663, Z -5.5000, A 0.000, B 0.000, C 0.000 }
gfCNCPoint4[14068] = {X 314.6073, Y 41.1790, Z -5.5000, A 0.000, B 0.000, C 0.000 }
gfCNCPoint4[14069] = {X 315.1932, Y 41.8054, Z -5.5000, A 0.000, B 0.000, C 0.000 }
gfCNCPoint4[14070] = {X 315.6321, Y 42.5424, Z -5.5000, A 0.000, B 0.000, C 0.000 }
gfCNCPoint4[14071] = {X 315.9038, Y 43.3560, Z -5.5000, A 0.000, B 0.000, C 0.000 }
gfCNCPoint4[14072] = {X 315.9957, Y 44.2089, Z -5.5000, A 0.000, B 0.000, C 0.000 }
gfCNCPoint4[14073] = {X 315.9957, Y 45.0000, Z -5.5000, A 0.000, B 0.000, C 0.000 }
gfCNCPoint4[14074] = {X 315.8954, Y 45.8901, Z -5.5000, A 0.000, B 0.000, C 0.000 }
gfCNCPoint4[14075] = {X 315.5996, Y 46.7355, Z -5.5000, A 0.000, B 0.000, C 0.000 }
gfCNCPoint4[14076] = {X 315.1230, Y 47.4940, Z -5.5000, A 0.000, B 0.000, C 0.000 }
gfCNCPoint4[14077] = {X 314.4897, Y 48.1273, Z -5.5000, A 0.000, B 0.000, C 0.000 }
gfCNCPoint4[14078] = {X 313.7313, Y 48.6039, Z -5.5000, A 0.000, B 0.000, C 0.000 }
gfCNCPoint4[14079] = {X 312.8858, Y 48.8997, Z -5.5000, A 0.000, B 0.000, C 0.000 }
gfCNCPoint4[14080] = {X 311.9957, Y 49.0000, Z -5.5000, A 0.000, B 0.000, C 0.000 }
gfCNCPoint4[14081] = {X 305.5523, Y 49.0000, Z -5.5000, A 0.000, B 0.000, C 0.000 }
gfCNCPoint4[14082] = {X 304.6622, Y 48.8997, Z -5.5000, A 0.000, B 0.000, C 0.000 }
gfCNCPoint4[14083] = {X 303.8167, Y 48.6039, Z -5.5000, A 0.000, B 0.000, C 0.000 }
gfCNCPoint4[14084] = {X 303.0583, Y 48.1273, Z -5.5000, A 0.000, B 0.000, C 0.000 }
gfCNCPoint4[14085] = {X 302.4249, Y 47.4939, Z -5.5000, A 0.000, B 0.000, C 0.000 }
gfCNCPoint4[14086] = {X 301.9484, Y 46.7355, Z -5.5000, A 0.000, B 0.000, C 0.000 }
gfCNCPoint4[14087] = {X 301.6525, Y 45.8901, Z -5.5000, A 0.000, B 0.000, C 0.000 }
gfCNCPoint4[14088] = {X 301.5523, Y 45.0000, Z -5.5000, A 0.000, B 0.000, C 0.000 }
gfCNCPoint4[14089] = {X 301.5523, Y 44.2089, Z -5.5000, A 0.000, B 0.000, C 0.000 }
gfCNCPoint4[14090] = {X 301.6696, Y 43.3029, Z -5.5000, A 0.000, B 0.000, C 0.000 }
gfCNCPoint4[14091] = {X 301.9734, Y 42.4414, Z -5.5000, A 0.000, B 0.000, C 0.000 }
gfCNCPoint4[14092] = {X 302.4504, Y 41.6623, Z -5.5000, A 0.000, B 0.000, C 0.000 }
gfCNCPoint4[14093] = {X 303.0794, Y 40.9999, Z -5.5000, A 0.000, B 0.000, C 0.000 }
gfCNCPoint4[14094] = {X 303.0794, Y 33.7143, Z -5.5000, A 0.000, B 0.000, C 0.000 }
gfCNCPoint4[14095] = {X 293.9347, Y 33.7143, Z -5.5000, A 0.000, B 0.000, C 0.000 }
gfCNCPoint4[14096] = {X 293.5347, Y 33.7141, Z -5.5000, A 0.000, B 0.000, C 0.000 }
gfCNCPoint4[14097] = {X 293.5340, Y 41.0518, Z -5.5000, A 0.000, B 0.000, C 0.000 }
gfCNCPoint4[14098] = {X 294.1713, Y 41.6932, Z -5.5000, A 0.000, B 0.000, C 0.000 }
gfCNCPoint4[14099] = {X 294.6524, Y 42.4587, Z -5.5000, A 0.000, B 0.000, C 0.000 }
gfCNCPoint4[14100] = {X 294.9539, Y 43.3111, Z -5.5000, A 0.000, B 0.000, C 0.000 }
gfCNCPoint4[14101] = {X 295.0611, Y 44.2089, Z -5.5000, A 0.000, B 0.000, C 0.000 }
gfCNCPoint4[14102] = {X 295.0611, Y 45.0000, Z -5.5000, A 0.000, B 0.000, C 0.000 }
gfCNCPoint4[14103] = {X 294.9608, Y 45.8901, Z -5.5000, A 0.000, B 0.000, C 0.000 }
gfCNCPoint4[14104] = {X 294.6650, Y 46.7355, Z -5.5000, A 0.000, B 0.000, C 0.000 }
gfCNCPoint4[14105] = {X 294.1885, Y 47.4940, Z -5.5000, A 0.000, B 0.000, C 0.000 }
gfCNCPoint4[14106] = {X 293.5551, Y 48.1273, Z -5.5000, A 0.000, B 0.000, C 0.000 }
gfCNCPoint4[14107] = {X 292.7967, Y 48.6039, Z -5.5000, A 0.000, B 0.000, C 0.000 }
gfCNCPoint4[14108] = {X 291.9512, Y 48.8997, Z -5.5000, A 0.000, B 0.000, C 0.000 }
gfCNCPoint4[14109] = {X 291.0611, Y 49.0000, Z -5.5000, A 0.000, B 0.000, C 0.000 }
gfCNCPoint4[14110] = {X 284.6177, Y 49.0000, Z -5.5000, A 0.000, B 0.000, C 0.000 }
gfCNCPoint4[14111] = {X 283.7276, Y 48.8997, Z -5.5000, A 0.000, B 0.000, C 0.000 }
gfCNCPoint4[14112] = {X 282.8821, Y 48.6039, Z -5.5000, A 0.000, B 0.000, C 0.000 }
gfCNCPoint4[14113] = {X 282.1237, Y 48.1273, Z -5.5000, A 0.000, B 0.000, C 0.000 }
gfCNCPoint4[14114] = {X 281.4903, Y 47.4939, Z -5.5000, A 0.000, B 0.000, C 0.000 }
gfCNCPoint4[14115] = {X 281.0138, Y 46.7355, Z -5.5000, A 0.000, B 0.000, C 0.000 }
gfCNCPoint4[14116] = {X 280.7180, Y 45.8901, Z -5.5000, A 0.000, B 0.000, C 0.000 }
gfCNCPoint4[14117] = {X 280.6177, Y 45.0000, Z -5.5000, A 0.000, B 0.000, C 0.000 }
gfCNCPoint4[14118] = {X 280.6177, Y 44.2089, Z -5.5000, A 0.000, B 0.000, C 0.000 }
gfCNCPoint4[14119] = {X 280.7227, Y 43.3125, Z -5.5000, A 0.000, B 0.000, C 0.000 }
gfCNCPoint4[14120] = {X 281.0237, Y 42.4616, Z -5.5000, A 0.000, B 0.000, C 0.000 }
gfCNCPoint4[14121] = {X 281.5058, Y 41.6986, Z -5.5000, A 0.000, B 0.000, C 0.000 }
gfCNCPoint4[14122] = {X 282.1450, Y 41.0615, Z -5.5000, A 0.000, B 0.000, C 0.000 }
gfCNCPoint4[14123] = {X 282.1448, Y 28.5922, Z -5.5000, A 0.000, B 0.000, C 0.000 }
gfCNCPoint4[14124] = {X 278.0648, Y 28.5923, Z -5.5000, A 0.000, B 0.000, C 0.000 }
gfCNCPoint4[14125] = {X 278.0648, Y 28.5923, Z -2.5000, A 0.000, B 0.000, C 0.000 }
gfCNCPoint4[14126] = {X 278.0648, Y 28.5923, Z 11.0000, A 0.000, B 0.000, C 0.000 }
gfCNCPoint4[14127] = {X 353.3539, Y 107.0409, Z 11.0000, A 0.000, B 0.000, C 0.000 }
gfCNCPoint4[14128] = {X 353.3539, Y 107.0409, Z -2.5000, A 0.000, B 0.000, C 0.000 }
gfCNCPoint4[14129] = {X 353.3539, Y 107.0409, Z -5.5000, A 0.000, B 0.000, C 0.000 }
gfCNCPoint4[14130] = {X 353.2425, Y 102.9624, Z -5.5000, A 0.000, B 0.000, C 0.000 }
gfCNCPoint4[14131] = {X 348.1838, Y 103.0323, Z -5.5000, A 0.000, B 0.000, C 0.000 }
gfCNCPoint4[14132] = {X 343.1250, Y 102.9655, Z -5.5000, A 0.000, B 0.000, C 0.000 }
gfCNCPoint4[14133] = {X 338.0700, Y 102.7621, Z -5.5000, A 0.000, B 0.000, C 0.000 }
gfCNCPoint4[14134] = {X 334.1157, Y 102.4852, Z -5.5000, A 0.000, B 0.000, C 0.000 }
gfCNCPoint4[14135] = {X 330.1764, Y 102.0433, Z -5.5000, A 0.000, B 0.000, C 0.000 }
gfCNCPoint4[14136] = {X 326.2590, Y 101.4373, Z -5.5000, A 0.000, B 0.000, C 0.000 }
gfCNCPoint4[14137] = {X 323.4093, Y 100.8330, Z -5.5000, A 0.000, B 0.000, C 0.000 }
gfCNCPoint4[14138] = {X 320.6119, Y 100.0201, Z -5.5000, A 0.000, B 0.000, C 0.000 }
gfCNCPoint4[14139] = {X 317.8821, Y 99.0029, Z -5.5000, A 0.000, B 0.000, C 0.000 }
gfCNCPoint4[14140] = {X 316.3692, Y 98.3052, Z -5.5000, A 0.000, B 0.000, C 0.000 }
gfCNCPoint4[14141] = {X 314.9199, Y 97.4834, Z -5.5000, A 0.000, B 0.000, C 0.000 }
gfCNCPoint4[14142] = {X 313.5445, Y 96.5432, Z -5.5000, A 0.000, B 0.000, C 0.000 }
gfCNCPoint4[14143] = {X 312.2525, Y 95.4913, Z -5.5000, A 0.000, B 0.000, C 0.000 }
gfCNCPoint4[14144] = {X 311.2488, Y 94.4927, Z -5.5000, A 0.000, B 0.000, C 0.000 }
gfCNCPoint4[14145] = {X 310.3705, Y 93.3822, Z -5.5000, A 0.000, B 0.000, C 0.000 }
gfCNCPoint4[14146] = {X 309.6301, Y 92.1755, Z -5.5000, A 0.000, B 0.000, C 0.000 }
gfCNCPoint4[14147] = {X 309.0379, Y 90.8895, Z -5.5000, A 0.000, B 0.000, C 0.000 }
gfCNCPoint4[14148] = {X 308.6023, Y 89.5423, Z -5.5000, A 0.000, B 0.000, C 0.000 }
gfCNCPoint4[14149] = {X 308.2588, Y 87.9192, Z -5.5000, A 0.000, B 0.000, C 0.000 }
gfCNCPoint4[14150] = {X 308.0559, Y 86.2727, Z -5.5000, A 0.000, B 0.000, C 0.000 }
gfCNCPoint4[14151] = {X 307.9950, Y 84.6147, Z -5.5000, A 0.000, B 0.000, C 0.000 }
gfCNCPoint4[14152] = {X 307.9963, Y 63.2122, Z -5.5000, A 0.000, B 0.000, C 0.000 }
gfCNCPoint4[14153] = {X 307.1448, Y 63.0029, Z -5.5000, A 0.000, B 0.000, C 0.000 }
gfCNCPoint4[14154] = {X 306.3531, Y 62.6261, Z -5.5000, A 0.000, B 0.000, C 0.000 }
gfCNCPoint4[14155] = {X 305.6538, Y 62.0971, Z -5.5000, A 0.000, B 0.000, C 0.000 }
gfCNCPoint4[14156] = {X 305.0758, Y 61.4378, Z -5.5000, A 0.000, B 0.000, C 0.000 }
gfCNCPoint4[14157] = {X 304.6427, Y 60.6754, Z -5.5000, A 0.000, B 0.000, C 0.000 }
gfCNCPoint4[14158] = {X 304.3726, Y 59.8413, Z -5.5000, A 0.000, B 0.000, C 0.000 }
gfCNCPoint4[14159] = {X 304.2764, Y 58.9697, Z -5.5000, A 0.000, B 0.000, C 0.000 }
gfCNCPoint4[14160] = {X 304.2762, Y 58.0000, Z -5.5000, A 0.000, B 0.000, C 0.000 }
gfCNCPoint4[14161] = {X 304.3845, Y 57.0387, Z -5.5000, A 0.000, B 0.000, C 0.000 }
gfCNCPoint4[14162] = {X 304.7040, Y 56.1256, Z -5.5000, A 0.000, B 0.000, C 0.000 }
gfCNCPoint4[14163] = {X 305.2187, Y 55.3065, Z -5.5000, A 0.000, B 0.000, C 0.000 }
gfCNCPoint4[14164] = {X 305.9027, Y 54.6225, Z -5.5000, A 0.000, B 0.000, C 0.000 }
gfCNCPoint4[14165] = {X 306.7218, Y 54.1078, Z -5.5000, A 0.000, B 0.000, C 0.000 }
gfCNCPoint4[14166] = {X 307.6349, Y 53.7883, Z -5.5000, A 0.000, B 0.000, C 0.000 }
gfCNCPoint4[14167] = {X 308.5962, Y 53.6800, Z -5.5000, A 0.000, B 0.000, C 0.000 }
gfCNCPoint4[14168] = {X 324.3107, Y 53.6800, Z -5.5000, A 0.000, B 0.000, C 0.000 }
gfCNCPoint4[14169] = {X 325.2720, Y 53.7883, Z -5.5000, A 0.000, B 0.000, C 0.000 }
gfCNCPoint4[14170] = {X 326.1851, Y 54.1078, Z -5.5000, A 0.000, B 0.000, C 0.000 }
gfCNCPoint4[14171] = {X 327.0042, Y 54.6225, Z -5.5000, A 0.000, B 0.000, C 0.000 }
gfCNCPoint4[14172] = {X 327.6882, Y 55.3065, Z -5.5000, A 0.000, B 0.000, C 0.000 }
gfCNCPoint4[14173] = {X 328.2029, Y 56.1256, Z -5.5000, A 0.000, B 0.000, C 0.000 }
gfCNCPoint4[14174] = {X 328.5224, Y 57.0387, Z -5.5000, A 0.000, B 0.000, C 0.000 }
gfCNCPoint4[14175] = {X 328.6307, Y 58.0000, Z -5.5000, A 0.000, B 0.000, C 0.000 }
gfCNCPoint4[14176] = {X 328.6307, Y 58.9359, Z -5.5000, A 0.000, B 0.000, C 0.000 }
gfCNCPoint4[14177] = {X 328.5367, Y 59.8122, Z -5.5000, A 0.000, B 0.000, C 0.000 }
gfCNCPoint4[14178] = {X 328.2683, Y 60.6517, Z -5.5000, A 0.000, B 0.000, C 0.000 }
gfCNCPoint4[14179] = {X 327.8365, Y 61.4200, Z -5.5000, A 0.000, B 0.000, C 0.000 }
gfCNCPoint4[14180] = {X 327.2590, Y 62.0857, Z -5.5000, A 0.000, B 0.000, C 0.000 }
gfCNCPoint4[14181] = {X 326.5593, Y 62.6216, Z -5.5000, A 0.000, B 0.000, C 0.000 }
gfCNCPoint4[14182] = {X 325.7661, Y 63.0058, Z -5.5000, A 0.000, B 0.000, C 0.000 }
gfCNCPoint4[14183] = {X 324.9118, Y 63.2226, Z -5.5000, A 0.000, B 0.000, C 0.000 }
gfCNCPoint4[14184] = {X 324.9136, Y 83.2295, Z -5.5000, A 0.000, B 0.000, C 0.000 }
gfCNCPoint4[14185] = {X 324.9271, Y 84.6147, Z -5.5000, A 0.000, B 0.000, C 0.000 }
gfCNCPoint4[14186] = {X 325.0045, Y 85.8498, Z -5.5000, A 0.000, B 0.000, C 0.000 }
gfCNCPoint4[14187] = {X 325.2262, Y 87.0673, Z -5.5000, A 0.000, B 0.000, C 0.000 }
gfCNCPoint4[14188] = {X 325.4716, Y 87.3359, Z -5.5000, A 0.000, B 0.000, C 0.000 }
gfCNCPoint4[14189] = {X 325.7737, Y 87.5385, Z -5.5000, A 0.000, B 0.000, C 0.000 }
gfCNCPoint4[14190] = {X 326.2249, Y 87.7937, Z -5.5000, A 0.000, B 0.000, C 0.000 }
gfCNCPoint4[14191] = {X 327.6626, Y 88.3902, Z -5.5000, A 0.000, B 0.000, C 0.000 }
gfCNCPoint4[14192] = {X 329.1569, Y 88.8257, Z -5.5000, A 0.000, B 0.000, C 0.000 }
gfCNCPoint4[14193] = {X 331.4311, Y 89.2991, Z -5.5000, A 0.000, B 0.000, C 0.000 }
gfCNCPoint4[14194] = {X 333.7258, Y 89.6603, Z -5.5000, A 0.000, B 0.000, C 0.000 }
gfCNCPoint4[14195] = {X 336.0355, Y 89.9083, Z -5.5000, A 0.000, B 0.000, C 0.000 }
gfCNCPoint4[14196] = {X 340.4056, Y 90.2026, Z -5.5000, A 0.000, B 0.000, C 0.000 }
gfCNCPoint4[14197] = {X 344.7828, Y 90.3564, Z -5.5000, A 0.000, B 0.000, C 0.000 }
gfCNCPoint4[14198] = {X 349.1628, Y 90.3697, Z -5.5000, A 0.000, B 0.000, C 0.000 }
gfCNCPoint4[14199] = {X 353.3143, Y 90.3014, Z -5.5000, A 0.000, B 0.000, C 0.000 }
gfCNCPoint4[14200] = {X 357.4607, Y 90.0824, Z -5.5000, A 0.000, B 0.000, C 0.000 }
gfCNCPoint4[14201] = {X 361.5963, Y 89.7130, Z -5.5000, A 0.000, B 0.000, C 0.000 }
gfCNCPoint4[14202] = {X 363.6775, Y 89.4259, Z -5.5000, A 0.000, B 0.000, C 0.000 }
gfCNCPoint4[14203] = {X 365.7397, Y 89.0239, Z -5.5000, A 0.000, B 0.000, C 0.000 }
gfCNCPoint4[14204] = {X 367.7763, Y 88.5083, Z -5.5000, A 0.000, B 0.000, C 0.000 }
gfCNCPoint4[14205] = {X 368.7083, Y 88.1950, Z -5.5000, A 0.000, B 0.000, C 0.000 }
gfCNCPoint4[14206] = {X 369.5993, Y 87.7793, Z -5.5000, A 0.000, B 0.000, C 0.000 }
gfCNCPoint4[14207] = {X 370.4380, Y 87.2662, Z -5.5000, A 0.000, B 0.000, C 0.000 }
gfCNCPoint4[14208] = {X 370.5877, Y 87.1104, Z -5.5000, A 0.000, B 0.000, C 0.000 }
gfCNCPoint4[14209] = {X 370.6649, Y 86.9086, Z -5.5000, A 0.000, B 0.000, C 0.000 }
gfCNCPoint4[14210] = {X 370.8560, Y 85.3738, Z -5.5000, A 0.000, B 0.000, C 0.000 }
gfCNCPoint4[14211] = {X 370.9197, Y 83.8285, Z -5.5000, A 0.000, B 0.000, C 0.000 }
gfCNCPoint4[14212] = {X 370.9203, Y 63.2123, Z -5.5000, A 0.000, B 0.000, C 0.000 }
gfCNCPoint4[14213] = {X 370.0686, Y 63.0032, Z -5.5000, A 0.000, B 0.000, C 0.000 }
gfCNCPoint4[14214] = {X 369.2768, Y 62.6264, Z -5.5000, A 0.000, B 0.000, C 0.000 }
gfCNCPoint4[14215] = {X 368.5773, Y 62.0975, Z -5.5000, A 0.000, B 0.000, C 0.000 }
gfCNCPoint4[14216] = {X 367.9991, Y 61.4382, Z -5.5000, A 0.000, B 0.000, C 0.000 }
gfCNCPoint4[14217] = {X 367.5659, Y 60.6757, Z -5.5000, A 0.000, B 0.000, C 0.000 }
gfCNCPoint4[14218] = {X 367.2956, Y 59.8414, Z -5.5000, A 0.000, B 0.000, C 0.000 }
gfCNCPoint4[14219] = {X 367.1994, Y 58.9697, Z -5.5000, A 0.000, B 0.000, C 0.000 }
gfCNCPoint4[14220] = {X 367.1993, Y 58.0000, Z -5.5000, A 0.000, B 0.000, C 0.000 }
gfCNCPoint4[14221] = {X 367.3076, Y 57.0387, Z -5.5000, A 0.000, B 0.000, C 0.000 }
gfCNCPoint4[14222] = {X 367.6271, Y 56.1256, Z -5.5000, A 0.000, B 0.000, C 0.000 }
gfCNCPoint4[14223] = {X 368.1418, Y 55.3065, Z -5.5000, A 0.000, B 0.000, C 0.000 }
gfCNCPoint4[14224] = {X 368.8258, Y 54.6225, Z -5.5000, A 0.000, B 0.000, C 0.000 }
gfCNCPoint4[14225] = {X 369.6449, Y 54.1078, Z -5.5000, A 0.000, B 0.000, C 0.000 }
gfCNCPoint4[14226] = {X 370.5580, Y 53.7883, Z -5.5000, A 0.000, B 0.000, C 0.000 }
gfCNCPoint4[14227] = {X 371.5193, Y 53.6800, Z -5.5000, A 0.000, B 0.000, C 0.000 }
gfCNCPoint4[14228] = {X 388.0597, Y 53.6800, Z -5.5000, A 0.000, B 0.000, C 0.000 }
gfCNCPoint4[14229] = {X 389.0210, Y 53.7883, Z -5.5000, A 0.000, B 0.000, C 0.000 }
gfCNCPoint4[14230] = {X 389.9341, Y 54.1078, Z -5.5000, A 0.000, B 0.000, C 0.000 }
gfCNCPoint4[14231] = {X 390.7532, Y 54.6225, Z -5.5000, A 0.000, B 0.000, C 0.000 }
gfCNCPoint4[14232] = {X 391.4372, Y 55.3065, Z -5.5000, A 0.000, B 0.000, C 0.000 }
gfCNCPoint4[14233] = {X 391.9519, Y 56.1256, Z -5.5000, A 0.000, B 0.000, C 0.000 }
gfCNCPoint4[14234] = {X 392.2714, Y 57.0387, Z -5.5000, A 0.000, B 0.000, C 0.000 }
gfCNCPoint4[14235] = {X 392.3797, Y 58.0000, Z -5.5000, A 0.000, B 0.000, C 0.000 }
gfCNCPoint4[14236] = {X 392.3797, Y 58.9342, Z -5.5000, A 0.000, B 0.000, C 0.000 }
gfCNCPoint4[14237] = {X 392.2667, Y 59.9158, Z -5.5000, A 0.000, B 0.000, C 0.000 }
gfCNCPoint4[14238] = {X 391.9336, Y 60.8460, Z -5.5000, A 0.000, B 0.000, C 0.000 }
gfCNCPoint4[14239] = {X 391.4909, Y 61.5609, Z -5.5000, A 0.000, B 0.000, C 0.000 }
gfCNCPoint4[14240] = {X 390.9187, Y 62.1770, Z -5.5000, A 0.000, B 0.000, C 0.000 }
gfCNCPoint4[14241] = {X 390.2386, Y 62.6714, Z -5.5000, A 0.000, B 0.000, C 0.000 }
gfCNCPoint4[14242] = {X 389.4759, Y 63.0254, Z -5.5000, A 0.000, B 0.000, C 0.000 }
gfCNCPoint4[14243] = {X 388.6593, Y 63.2258, Z -5.5000, A 0.000, B 0.000, C 0.000 }
gfCNCPoint4[14244] = {X 388.6573, Y 84.6147, Z -5.5000, A 0.000, B 0.000, C 0.000 }
gfCNCPoint4[14245] = {X 388.5974, Y 86.2731, Z -5.5000, A 0.000, B 0.000, C 0.000 }
gfCNCPoint4[14246] = {X 388.3930, Y 87.9199, Z -5.5000, A 0.000, B 0.000, C 0.000 }
gfCNCPoint4[14247] = {X 388.0458, Y 89.5426, Z -5.5000, A 0.000, B 0.000, C 0.000 }
gfCNCPoint4[14248] = {X 387.5136, Y 91.1298, Z -5.5000, A 0.000, B 0.000, C 0.000 }
gfCNCPoint4[14249] = {X 386.7640, Y 92.6268, Z -5.5000, A 0.000, B 0.000, C 0.000 }
gfCNCPoint4[14250] = {X 385.8120, Y 94.0038, Z -5.5000, A 0.000, B 0.000, C 0.000 }
gfCNCPoint4[14251] = {X 384.6762, Y 95.2338, Z -5.5000, A 0.000, B 0.000, C 0.000 }
gfCNCPoint4[14252] = {X 383.1617, Y 96.5100, Z -5.5000, A 0.000, B 0.000, C 0.000 }
gfCNCPoint4[14253] = {X 381.5202, Y 97.6183, Z -5.5000, A 0.000, B 0.000, C 0.000 }
gfCNCPoint4[14254] = {X 379.7703, Y 98.5459, Z -5.5000, A 0.000, B 0.000, C 0.000 }
gfCNCPoint4[14255] = {X 377.4988, Y 99.5009, Z -5.5000, A 0.000, B 0.000, C 0.000 }
gfCNCPoint4[14256] = {X 375.1648, Y 100.2911, Z -5.5000, A 0.000, B 0.000, C 0.000 }
gfCNCPoint4[14257] = {X 372.7804, Y 100.9126, Z -5.5000, A 0.000, B 0.000, C 0.000 }
gfCNCPoint4[14258] = {X 368.8697, Y 101.6667, Z -5.5000, A 0.000, B 0.000, C 0.000 }
gfCNCPoint4[14259] = {X 364.9265, Y 102.2270, Z -5.5000, A 0.000, B 0.000, C 0.000 }
gfCNCPoint4[14260] = {X 360.9605, Y 102.5921, Z -5.5000, A 0.000, B 0.000, C 0.000 }
gfCNCPoint4[14261] = {X 357.1034, Y 102.8171, Z -5.5000, A 0.000, B 0.000, C 0.000 }
gfCNCPoint4[14262] = {X 353.2425, Y 102.9624, Z -5.5000, A 0.000, B 0.000, C 0.000 }
gfCNCPoint4[14263] = {X 353.3517, Y 106.9609, Z -5.5000, A 0.000, B 0.000, C 0.000 }
gfCNCPoint4[14264] = {X 353.2403, Y 102.8824, Z -5.5000, A 0.000, B 0.000, C 0.000 }
gfCNCPoint4[14265] = {X 348.1837, Y 102.9523, Z -5.5000, A 0.000, B 0.000, C 0.000 }
gfCNCPoint4[14266] = {X 343.1271, Y 102.8855, Z -5.5000, A 0.000, B 0.000, C 0.000 }
gfCNCPoint4[14267] = {X 338.0741, Y 102.6823, Z -5.5000, A 0.000, B 0.000, C 0.000 }
gfCNCPoint4[14268] = {X 334.1231, Y 102.4055, Z -5.5000, A 0.000, B 0.000, C 0.000 }
gfCNCPoint4[14269] = {X 330.1870, Y 101.9640, Z -5.5000, A 0.000, B 0.000, C 0.000 }
gfCNCPoint4[14270] = {X 326.2728, Y 101.3585, Z -5.5000, A 0.000, B 0.000, C 0.000 }
gfCNCPoint4[14271] = {X 323.4288, Y 100.7554, Z -5.5000, A 0.000, B 0.000, C 0.000 }
gfCNCPoint4[14272] = {X 320.6370, Y 99.9441, Z -5.5000, A 0.000, B 0.000, C 0.000 }
gfCNCPoint4[14273] = {X 317.9127, Y 98.9290, Z -5.5000, A 0.000, B 0.000, C 0.000 }
gfCNCPoint4[14274] = {X 316.4058, Y 98.2341, Z -5.5000, A 0.000, B 0.000, C 0.000 }
gfCNCPoint4[14275] = {X 314.9623, Y 97.4156, Z -5.5000, A 0.000, B 0.000, C 0.000 }
gfCNCPoint4[14276] = {X 313.5924, Y 96.4791, Z -5.5000, A 0.000, B 0.000, C 0.000 }
gfCNCPoint4[14277] = {X 312.3056, Y 95.4314, Z -5.5000, A 0.000, B 0.000, C 0.000 }
gfCNCPoint4[14278] = {X 311.3086, Y 94.4395, Z -5.5000, A 0.000, B 0.000, C 0.000 }
gfCNCPoint4[14279] = {X 310.4362, Y 93.3365, Z -5.5000, A 0.000, B 0.000, C 0.000 }
gfCNCPoint4[14280] = {X 309.7007, Y 92.1378, Z -5.5000, A 0.000, B 0.000, C 0.000 }
gfCNCPoint4[14281] = {X 309.1124, Y 90.8604, Z -5.5000, A 0.000, B 0.000, C 0.000 }
gfCNCPoint4[14282] = {X 308.6798, Y 89.5223, Z -5.5000, A 0.000, B 0.000, C 0.000 }
gfCNCPoint4[14283] = {X 308.3377, Y 87.9059, Z -5.5000, A 0.000, B 0.000, C 0.000 }
gfCNCPoint4[14284] = {X 308.1357, Y 86.2661, Z -5.5000, A 0.000, B 0.000, C 0.000 }
gfCNCPoint4[14285] = {X 308.0750, Y 84.6150, Z -5.5000, A 0.000, B 0.000, C 0.000 }
gfCNCPoint4[14286] = {X 308.0763, Y 63.1421, Z -5.5000, A 0.000, B 0.000, C 0.000 }
gfCNCPoint4[14287] = {X 307.2279, Y 62.9472, Z -5.5000, A 0.000, B 0.000, C 0.000 }
gfCNCPoint4[14288] = {X 306.4372, Y 62.5832, Z -5.5000, A 0.000, B 0.000, C 0.000 }
gfCNCPoint4[14289] = {X 305.7375, Y 62.0654, Z -5.5000, A 0.000, B 0.000, C 0.000 }
gfCNCPoint4[14290] = {X 305.1583, Y 61.4157, Z -5.5000, A 0.000, B 0.000, C 0.000 }
gfCNCPoint4[14291] = {X 304.7240, Y 60.6613, Z -5.5000, A 0.000, B 0.000, C 0.000 }
gfCNCPoint4[14292] = {X 304.4529, Y 59.8342, Z -5.5000, A 0.000, B 0.000, C 0.000 }
gfCNCPoint4[14293] = {X 304.3564, Y 58.9691, Z -5.5000, A 0.000, B 0.000, C 0.000 }
gfCNCPoint4[14294] = {X 304.3562, Y 58.0000, Z -5.5000, A 0.000, B 0.000, C 0.000 }
gfCNCPoint4[14295] = {X 304.4625, Y 57.0565, Z -5.5000, A 0.000, B 0.000, C 0.000 }
gfCNCPoint4[14296] = {X 304.7761, Y 56.1603, Z -5.5000, A 0.000, B 0.000, C 0.000 }
gfCNCPoint4[14297] = {X 305.2813, Y 55.3564, Z -5.5000, A 0.000, B 0.000, C 0.000 }
gfCNCPoint4[14298] = {X 305.9526, Y 54.6850, Z -5.5000, A 0.000, B 0.000, C 0.000 }
gfCNCPoint4[14299] = {X 306.7566, Y 54.1799, Z -5.5000, A 0.000, B 0.000, C 0.000 }
gfCNCPoint4[14300] = {X 307.6527, Y 53.8663, Z -5.5000, A 0.000, B 0.000, C 0.000 }
gfCNCPoint4[14301] = {X 308.5962, Y 53.7600, Z -5.5000, A 0.000, B 0.000, C 0.000 }
gfCNCPoint4[14302] = {X 324.3107, Y 53.7600, Z -5.5000, A 0.000, B 0.000, C 0.000 }
gfCNCPoint4[14303] = {X 325.2542, Y 53.8663, Z -5.5000, A 0.000, B 0.000, C 0.000 }
gfCNCPoint4[14304] = {X 326.1504, Y 54.1799, Z -5.5000, A 0.000, B 0.000, C 0.000 }
gfCNCPoint4[14305] = {X 326.9543, Y 54.6850, Z -5.5000, A 0.000, B 0.000, C 0.000 }
gfCNCPoint4[14306] = {X 327.6257, Y 55.3564, Z -5.5000, A 0.000, B 0.000, C 0.000 }
gfCNCPoint4[14307] = {X 328.1308, Y 56.1603, Z -5.5000, A 0.000, B 0.000, C 0.000 }
gfCNCPoint4[14308] = {X 328.4444, Y 57.0565, Z -5.5000, A 0.000, B 0.000, C 0.000 }
gfCNCPoint4[14309] = {X 328.5507, Y 58.0000, Z -5.5000, A 0.000, B 0.000, C 0.000 }
gfCNCPoint4[14310] = {X 328.5507, Y 58.9354, Z -5.5000, A 0.000, B 0.000, C 0.000 }
gfCNCPoint4[14311] = {X 328.4564, Y 59.8053, Z -5.5000, A 0.000, B 0.000, C 0.000 }
gfCNCPoint4[14312] = {X 328.1870, Y 60.6378, Z -5.5000, A 0.000, B 0.000, C 0.000 }
gfCNCPoint4[14313] = {X 327.7540, Y 61.3980, Z -5.5000, A 0.000, B 0.000, C 0.000 }
gfCNCPoint4[14314] = {X 327.1753, Y 62.0543, Z -5.5000, A 0.000, B 0.000, C 0.000 }
gfCNCPoint4[14315] = {X 326.4752, Y 62.5791, Z -5.5000, A 0.000, B 0.000, C 0.000 }
gfCNCPoint4[14316] = {X 325.6830, Y 62.9505, Z -5.5000, A 0.000, B 0.000, C 0.000 }
gfCNCPoint4[14317] = {X 324.8318, Y 63.1530, Z -5.5000, A 0.000, B 0.000, C 0.000 }
gfCNCPoint4[14318] = {X 324.8336, Y 83.2300, Z -5.5000, A 0.000, B 0.000, C 0.000 }
gfCNCPoint4[14319] = {X 324.8471, Y 84.6150, Z -5.5000, A 0.000, B 0.000, C 0.000 }
gfCNCPoint4[14320] = {X 324.9261, Y 85.8671, Z -5.5000, A 0.000, B 0.000, C 0.000 }
gfCNCPoint4[14321] = {X 325.1521, Y 87.1011, Z -5.5000, A 0.000, B 0.000, C 0.000 }
gfCNCPoint4[14322] = {X 325.4128, Y 87.3908, Z -5.5000, A 0.000, B 0.000, C 0.000 }
gfCNCPoint4[14323] = {X 325.7358, Y 87.6090, Z -5.5000, A 0.000, B 0.000, C 0.000 }
gfCNCPoint4[14324] = {X 326.1879, Y 87.8647, Z -5.5000, A 0.000, B 0.000, C 0.000 }
gfCNCPoint4[14325] = {X 327.6348, Y 88.4652, Z -5.5000, A 0.000, B 0.000, C 0.000 }
gfCNCPoint4[14326] = {X 329.1387, Y 88.9036, Z -5.5000, A 0.000, B 0.000, C 0.000 }
gfCNCPoint4[14327] = {X 331.4168, Y 89.3778, Z -5.5000, A 0.000, B 0.000, C 0.000 }
gfCNCPoint4[14328] = {X 333.7153, Y 89.7396, Z -5.5000, A 0.000, B 0.000, C 0.000 }
gfCNCPoint4[14329] = {X 336.0289, Y 89.9880, Z -5.5000, A 0.000, B 0.000, C 0.000 }
gfCNCPoint4[14330] = {X 340.4015, Y 90.2825, Z -5.5000, A 0.000, B 0.000, C 0.000 }
gfCNCPoint4[14331] = {X 344.7813, Y 90.4364, Z -5.5000, A 0.000, B 0.000, C 0.000 }
gfCNCPoint4[14332] = {X 349.1638, Y 90.4497, Z -5.5000, A 0.000, B 0.000, C 0.000 }
gfCNCPoint4[14333] = {X 353.3179, Y 90.3813, Z -5.5000, A 0.000, B 0.000, C 0.000 }
gfCNCPoint4[14334] = {X 357.4668, Y 90.1621, Z -5.5000, A 0.000, B 0.000, C 0.000 }
gfCNCPoint4[14335] = {X 361.6050, Y 89.7926, Z -5.5000, A 0.000, B 0.000, C 0.000 }
gfCNCPoint4[14336] = {X 363.6906, Y 89.5049, Z -5.5000, A 0.000, B 0.000, C 0.000 }
gfCNCPoint4[14337] = {X 365.7571, Y 89.1020, Z -5.5000, A 0.000, B 0.000, C 0.000 }
gfCNCPoint4[14338] = {X 367.7981, Y 88.5853, Z -5.5000, A 0.000, B 0.000, C 0.000 }
gfCNCPoint4[14339] = {X 368.7384, Y 88.2692, Z -5.5000, A 0.000, B 0.000, C 0.000 }
gfCNCPoint4[14340] = {X 369.6373, Y 87.8496, Z -5.5000, A 0.000, B 0.000, C 0.000 }
gfCNCPoint4[14341] = {X 370.4835, Y 87.3320, Z -5.5000, A 0.000, B 0.000, C 0.000 }
gfCNCPoint4[14342] = {X 370.6553, Y 87.1533, Z -5.5000, A 0.000, B 0.000, C 0.000 }
gfCNCPoint4[14343] = {X 370.7438, Y 86.9218, Z -5.5000, A 0.000, B 0.000, C 0.000 }
gfCNCPoint4[14344] = {X 370.9357, Y 85.3804, Z -5.5000, A 0.000, B 0.000, C 0.000 }
gfCNCPoint4[14345] = {X 370.9997, Y 83.8285, Z -5.5000, A 0.000, B 0.000, C 0.000 }
gfCNCPoint4[14346] = {X 371.0003, Y 63.1422, Z -5.5000, A 0.000, B 0.000, C 0.000 }
gfCNCPoint4[14347] = {X 370.1518, Y 62.9475, Z -5.5000, A 0.000, B 0.000, C 0.000 }
gfCNCPoint4[14348] = {X 369.3609, Y 62.5836, Z -5.5000, A 0.000, B 0.000, C 0.000 }
gfCNCPoint4[14349] = {X 368.6610, Y 62.0658, Z -5.5000, A 0.000, B 0.000, C 0.000 }
gfCNCPoint4[14350] = {X 368.0816, Y 61.4160, Z -5.5000, A 0.000, B 0.000, C 0.000 }
gfCNCPoint4[14351] = {X 367.6472, Y 60.6616, Z -5.5000, A 0.000, B 0.000, C 0.000 }
gfCNCPoint4[14352] = {X 367.3760, Y 59.8343, Z -5.5000, A 0.000, B 0.000, C 0.000 }
gfCNCPoint4[14353] = {X 367.2794, Y 58.9691, Z -5.5000, A 0.000, B 0.000, C 0.000 }
gfCNCPoint4[14354] = {X 367.2793, Y 58.0000, Z -5.5000, A 0.000, B 0.000, C 0.000 }
gfCNCPoint4[14355] = {X 367.3856, Y 57.0565, Z -5.5000, A 0.000, B 0.000, C 0.000 }
gfCNCPoint4[14356] = {X 367.6992, Y 56.1603, Z -5.5000, A 0.000, B 0.000, C 0.000 }
gfCNCPoint4[14357] = {X 368.2043, Y 55.3564, Z -5.5000, A 0.000, B 0.000, C 0.000 }
gfCNCPoint4[14358] = {X 368.8757, Y 54.6850, Z -5.5000, A 0.000, B 0.000, C 0.000 }
gfCNCPoint4[14359] = {X 369.6796, Y 54.1799, Z -5.5000, A 0.000, B 0.000, C 0.000 }
gfCNCPoint4[14360] = {X 370.5758, Y 53.8663, Z -5.5000, A 0.000, B 0.000, C 0.000 }
gfCNCPoint4[14361] = {X 371.5193, Y 53.7600, Z -5.5000, A 0.000, B 0.000, C 0.000 }
gfCNCPoint4[14362] = {X 388.0597, Y 53.7600, Z -5.5000, A 0.000, B 0.000, C 0.000 }
gfCNCPoint4[14363] = {X 389.0032, Y 53.8663, Z -5.5000, A 0.000, B 0.000, C 0.000 }
gfCNCPoint4[14364] = {X 389.8993, Y 54.1799, Z -5.5000, A 0.000, B 0.000, C 0.000 }
gfCNCPoint4[14365] = {X 390.7033, Y 54.6850, Z -5.5000, A 0.000, B 0.000, C 0.000 }
gfCNCPoint4[14366] = {X 391.3746, Y 55.3564, Z -5.5000, A 0.000, B 0.000, C 0.000 }
gfCNCPoint4[14367] = {X 391.8798, Y 56.1603, Z -5.5000, A 0.000, B 0.000, C 0.000 }
gfCNCPoint4[14368] = {X 392.1934, Y 57.0565, Z -5.5000, A 0.000, B 0.000, C 0.000 }
gfCNCPoint4[14369] = {X 392.2997, Y 58.0000, Z -5.5000, A 0.000, B 0.000, C 0.000 }
gfCNCPoint4[14370] = {X 392.2997, Y 58.9342, Z -5.5000, A 0.000, B 0.000, C 0.000 }
gfCNCPoint4[14371] = {X 392.1887, Y 59.8976, Z -5.5000, A 0.000, B 0.000, C 0.000 }
gfCNCPoint4[14372] = {X 391.8618, Y 60.8106, Z -5.5000, A 0.000, B 0.000, C 0.000 }
gfCNCPoint4[14373] = {X 391.4189, Y 61.5233, Z -5.5000, A 0.000, B 0.000, C 0.000 }
gfCNCPoint4[14374] = {X 390.8449, Y 62.1354, Z -5.5000, A 0.000, B 0.000, C 0.000 }
gfCNCPoint4[14375] = {X 390.1622, Y 62.6233, Z -5.5000, A 0.000, B 0.000, C 0.000 }
gfCNCPoint4[14376] = {X 389.3971, Y 62.9679, Z -5.5000, A 0.000, B 0.000, C 0.000 }
gfCNCPoint4[14377] = {X 388.5793, Y 63.1560, Z -5.5000, A 0.000, B 0.000, C 0.000 }
gfCNCPoint4[14378] = {X 388.5773, Y 84.6150, Z -5.5000, A 0.000, B 0.000, C 0.000 }
gfCNCPoint4[14379] = {X 388.5176, Y 86.2665, Z -5.5000, A 0.000, B 0.000, C 0.000 }
gfCNCPoint4[14380] = {X 388.3141, Y 87.9065, Z -5.5000, A 0.000, B 0.000, C 0.000 }
gfCNCPoint4[14381] = {X 387.9684, Y 89.5224, Z -5.5000, A 0.000, B 0.000, C 0.000 }
gfCNCPoint4[14382] = {X 387.4398, Y 91.0991, Z -5.5000, A 0.000, B 0.000, C 0.000 }
gfCNCPoint4[14383] = {X 386.6952, Y 92.5860, Z -5.5000, A 0.000, B 0.000, C 0.000 }
gfCNCPoint4[14384] = {X 385.7495, Y 93.9538, Z -5.5000, A 0.000, B 0.000, C 0.000 }
gfCNCPoint4[14385] = {X 384.6214, Y 95.1755, Z -5.5000, A 0.000, B 0.000, C 0.000 }
gfCNCPoint4[14386] = {X 383.1134, Y 96.4462, Z -5.5000, A 0.000, B 0.000, C 0.000 }
gfCNCPoint4[14387] = {X 381.4790, Y 97.5497, Z -5.5000, A 0.000, B 0.000, C 0.000 }
gfCNCPoint4[14388] = {X 379.7366, Y 98.4733, Z -5.5000, A 0.000, B 0.000, C 0.000 }
gfCNCPoint4[14389] = {X 377.4704, Y 99.4261, Z -5.5000, A 0.000, B 0.000, C 0.000 }
gfCNCPoint4[14390] = {X 375.1419, Y 100.2145, Z -5.5000, A 0.000, B 0.000, C 0.000 }
gfCNCPoint4[14391] = {X 372.7630, Y 100.8345, Z -5.5000, A 0.000, B 0.000, C 0.000 }
gfCNCPoint4[14392] = {X 368.8562, Y 101.5878, Z -5.5000, A 0.000, B 0.000, C 0.000 }
gfCNCPoint4[14393] = {X 364.9170, Y 102.1475, Z -5.5000, A 0.000, B 0.000, C 0.000 }
gfCNCPoint4[14394] = {X 360.9550, Y 102.5123, Z -5.5000, A 0.000, B 0.000, C 0.000 }
gfCNCPoint4[14395] = {X 357.0996, Y 102.7372, Z -5.5000, A 0.000, B 0.000, C 0.000 }
gfCNCPoint4[14396] = {X 353.2403, Y 102.8824, Z -5.5000, A 0.000, B 0.000, C 0.000 }
gfCNCPoint4[14397] = {X 353.3495, Y 106.8809, Z -5.5000, A 0.000, B 0.000, C 0.000 }
gfCNCPoint4[14398] = {X 353.2381, Y 102.8025, Z -5.5000, A 0.000, B 0.000, C 0.000 }
gfCNCPoint4[14399] = {X 348.1837, Y 102.8723, Z -5.5000, A 0.000, B 0.000, C 0.000 }
gfCNCPoint4[14400] = {X 343.1291, Y 102.8056, Z -5.5000, A 0.000, B 0.000, C 0.000 }
gfCNCPoint4[14401] = {X 338.0783, Y 102.6024, Z -5.5000, A 0.000, B 0.000, C 0.000 }
gfCNCPoint4[14402] = {X 334.1304, Y 102.3259, Z -5.5000, A 0.000, B 0.000, C 0.000 }
gfCNCPoint4[14403] = {X 330.1976, Y 101.8848, Z -5.5000, A 0.000, B 0.000, C 0.000 }
gfCNCPoint4[14404] = {X 326.2866, Y 101.2797, Z -5.5000, A 0.000, B 0.000, C 0.000 }
gfCNCPoint4[14405] = {X 323.4483, Y 100.6778, Z -5.5000, A 0.000, B 0.000, C 0.000 }
gfCNCPoint4[14406] = {X 320.6622, Y 99.8682, Z -5.5000, A 0.000, B 0.000, C 0.000 }
gfCNCPoint4[14407] = {X 317.9434, Y 98.8551, Z -5.5000, A 0.000, B 0.000, C 0.000 }
gfCNCPoint4[14408] = {X 316.4425, Y 98.1630, Z -5.5000, A 0.000, B 0.000, C 0.000 }
gfCNCPoint4[14409] = {X 315.0048, Y 97.3477, Z -5.5000, A 0.000, B 0.000, C 0.000 }
gfCNCPoint4[14410] = {X 313.6403, Y 96.4151, Z -5.5000, A 0.000, B 0.000, C 0.000 }
gfCNCPoint4[14411] = {X 312.3586, Y 95.3715, Z -5.5000, A 0.000, B 0.000, C 0.000 }
gfCNCPoint4[14412] = {X 311.3683, Y 94.3864, Z -5.5000, A 0.000, B 0.000, C 0.000 }
gfCNCPoint4[14413] = {X 310.5018, Y 93.2907, Z -5.5000, A 0.000, B 0.000, C 0.000 }
gfCNCPoint4[14414] = {X 309.7712, Y 92.1001, Z -5.5000, A 0.000, B 0.000, C 0.000 }
gfCNCPoint4[14415] = {X 309.1870, Y 90.8313, Z -5.5000, A 0.000, B 0.000, C 0.000 }
gfCNCPoint4[14416] = {X 308.7572, Y 89.5022, Z -5.5000, A 0.000, B 0.000, C 0.000 }
gfCNCPoint4[14417] = {X 308.4166, Y 87.8925, Z -5.5000, A 0.000, B 0.000, C 0.000 }
gfCNCPoint4[14418] = {X 308.2154, Y 86.2596, Z -5.5000, A 0.000, B 0.000, C 0.000 }
gfCNCPoint4[14419] = {X 308.1550, Y 84.6153, Z -5.5000, A 0.000, B 0.000, C 0.000 }
gfCNCPoint4[14420] = {X 308.1563, Y 63.0707, Z -5.5000, A 0.000, B 0.000, C 0.000 }
gfCNCPoint4[14421] = {X 307.3112, Y 62.8906, Z -5.5000, A 0.000, B 0.000, C 0.000 }
gfCNCPoint4[14422] = {X 306.5216, Y 62.5398, Z -5.5000, A 0.000, B 0.000, C 0.000 }
gfCNCPoint4[14423] = {X 305.8214, Y 62.0334, Z -5.5000, A 0.000, B 0.000, C 0.000 }
gfCNCPoint4[14424] = {X 305.2410, Y 61.3933, Z -5.5000, A 0.000, B 0.000, C 0.000 }
gfCNCPoint4[14425] = {X 304.8053, Y 60.6471, Z -5.5000, A 0.000, B 0.000, C 0.000 }
gfCNCPoint4[14426] = {X 304.5332, Y 59.8270, Z -5.5000, A 0.000, B 0.000, C 0.000 }
gfCNCPoint4[14427] = {X 304.4364, Y 58.9684, Z -5.5000, A 0.000, B 0.000, C 0.000 }
gfCNCPoint4[14428] = {X 304.4362, Y 58.0000, Z -5.5000, A 0.000, B 0.000, C 0.000 }
gfCNCPoint4[14429] = {X 304.5405, Y 57.0743, Z -5.5000, A 0.000, B 0.000, C 0.000 }
gfCNCPoint4[14430] = {X 304.8482, Y 56.1950, Z -5.5000, A 0.000, B 0.000, C 0.000 }
gfCNCPoint4[14431] = {X 305.3438, Y 55.4063, Z -5.5000, A 0.000, B 0.000, C 0.000 }
gfCNCPoint4[14432] = {X 306.0025, Y 54.7476, Z -5.5000, A 0.000, B 0.000, C 0.000 }
gfCNCPoint4[14433] = {X 306.7913, Y 54.2520, Z -5.5000, A 0.000, B 0.000, C 0.000 }
gfCNCPoint4[14434] = {X 307.6705, Y 53.9443, Z -5.5000, A 0.000, B 0.000, C 0.000 }
gfCNCPoint4[14435] = {X 308.5962, Y 53.8400, Z -5.5000, A 0.000, B 0.000, C 0.000 }
gfCNCPoint4[14436] = {X 324.3107, Y 53.8400, Z -5.5000, A 0.000, B 0.000, C 0.000 }
gfCNCPoint4[14437] = {X 325.2364, Y 53.9443, Z -5.5000, A 0.000, B 0.000, C 0.000 }
gfCNCPoint4[14438] = {X 326.1156, Y 54.2520, Z -5.5000, A 0.000, B 0.000, C 0.000 }
gfCNCPoint4[14439] = {X 326.9044, Y 54.7476, Z -5.5000, A 0.000, B 0.000, C 0.000 }
gfCNCPoint4[14440] = {X 327.5631, Y 55.4063, Z -5.5000, A 0.000, B 0.000, C 0.000 }
gfCNCPoint4[14441] = {X 328.0587, Y 56.1950, Z -5.5000, A 0.000, B 0.000, C 0.000 }
gfCNCPoint4[14442] = {X 328.3664, Y 57.0743, Z -5.5000, A 0.000, B 0.000, C 0.000 }
gfCNCPoint4[14443] = {X 328.4707, Y 58.0000, Z -5.5000, A 0.000, B 0.000, C 0.000 }
gfCNCPoint4[14444] = {X 328.4707, Y 58.9350, Z -5.5000, A 0.000, B 0.000, C 0.000 }
gfCNCPoint4[14445] = {X 328.3760, Y 59.7984, Z -5.5000, A 0.000, B 0.000, C 0.000 }
gfCNCPoint4[14446] = {X 328.1057, Y 60.6238, Z -5.5000, A 0.000, B 0.000, C 0.000 }
gfCNCPoint4[14447] = {X 327.6714, Y 61.3759, Z -5.5000, A 0.000, B 0.000, C 0.000 }
gfCNCPoint4[14448] = {X 327.0915, Y 62.0226, Z -5.5000, A 0.000, B 0.000, C 0.000 }
gfCNCPoint4[14449] = {X 326.3910, Y 62.5360, Z -5.5000, A 0.000, B 0.000, C 0.000 }
gfCNCPoint4[14450] = {X 325.5998, Y 62.8944, Z -5.5000, A 0.000, B 0.000, C 0.000 }
gfCNCPoint4[14451] = {X 324.7518, Y 63.0822, Z -5.5000, A 0.000, B 0.000, C 0.000 }
gfCNCPoint4[14452] = {X 324.7536, Y 83.2304, Z -5.5000, A 0.000, B 0.000, C 0.000 }
gfCNCPoint4[14453] = {X 324.7671, Y 84.6153, Z -5.5000, A 0.000, B 0.000, C 0.000 }
gfCNCPoint4[14454] = {X 324.8476, Y 85.8842, Z -5.5000, A 0.000, B 0.000, C 0.000 }
gfCNCPoint4[14455] = {X 325.0779, Y 87.1345, Z -5.5000, A 0.000, B 0.000, C 0.000 }
gfCNCPoint4[14456] = {X 325.3539, Y 87.4456, Z -5.5000, A 0.000, B 0.000, C 0.000 }
gfCNCPoint4[14457] = {X 325.6979, Y 87.6795, Z -5.5000, A 0.000, B 0.000, C 0.000 }
gfCNCPoint4[14458] = {X 326.1508, Y 87.9356, Z -5.5000, A 0.000, B 0.000, C 0.000 }
gfCNCPoint4[14459] = {X 327.6069, Y 88.5402, Z -5.5000, A 0.000, B 0.000, C 0.000 }
gfCNCPoint4[14460] = {X 329.1206, Y 88.9815, Z -5.5000, A 0.000, B 0.000, C 0.000 }
gfCNCPoint4[14461] = {X 331.4025, Y 89.4565, Z -5.5000, A 0.000, B 0.000, C 0.000 }
gfCNCPoint4[14462] = {X 333.7049, Y 89.8189, Z -5.5000, A 0.000, B 0.000, C 0.000 }
gfCNCPoint4[14463] = {X 336.0223, Y 90.0677, Z -5.5000, A 0.000, B 0.000, C 0.000 }
